; move to the rack
TRIGGER WHEN DISTANCE=1 DELAY=-1 DO Schrittmerker_R1Place(10150,10002,FPlace_R1_L2_S4_VP1,XPlace_R1_L2_S4_VP1) PRIO=-1
;FOLD PTP Place_R1_L2_S4_VP1 CONT Vel=12 % PPlace_R1_L2_S4_VP1 Tool[2]:Lower Gripper Base[0];%{PE}%R8.3.21,%MKUKATPBASIS,%CMOVE,%VPTP,%P 1:PTP, 2:Place_R1_L2_S4_VP1, 3:C_DIS, 5:12, 7:PPlace_R1_L2_S4_VP1
$BWDSTART=FALSE
PDAT_ACT= PPPlace_R1_L2_S4_VP1
FDAT_ACT= FPlace_R1_L2_S4_VP1
BAS(#PTP_PARAMS,12)
PTP XPlace_R1_L2_S4_VP1 C_DIS
;ENDFOLD
TRIGGER WHEN DISTANCE=1 DELAY=-1 DO Schrittmerker_R1Place(10151,10150,FPlace_R1_L2_S4_VP2,XPlace_R1_L2_S4_VP2) PRIO=-1
;FOLD PTP Place_R1_L2_S4_VP2 CONT Vel=12 % PPlace_R1_L2_S4_VP2 Tool[2]:Lower Gripper Base[0];%{PE}%R8.3.21,%MKUKATPBASIS,%CMOVE,%VPTP,%P 1:PTP, 2:Place_R1_L2_S4_VP2, 3:C_DIS, 5:12, 7:PPlace_R1_L2_S4_VP2
$BWDSTART=FALSE
PDAT_ACT= PPPlace_R1_L2_S4_VP2
FDAT_ACT= FPlace_R1_L2_S4_VP2
BAS(#PTP_PARAMS,12)
PTP XPlace_R1_L2_S4_VP2 C_DIS
;ENDFOLD
TRIGGER WHEN DISTANCE=1 DELAY=-1 DO Schrittmerker_R1Place(10152,10151,FPlace_R1_L2_S4_VP3,XPlace_R1_L2_S4_VP3) PRIO=-1
;FOLD PTP Place_R1_L2_S4_VP3 CONT Vel=12 % PPlace_R1_L2_S4_VP3 Tool[2]:Lower Gripper Base[0];%{PE}%R8.3.21,%MKUKATPBASIS,%CMOVE,%VPTP,%P 1:PTP, 2:Place_R1_L2_S4_VP3, 3:C_DIS, 5:12, 7:PPlace_R1_L2_S4_VP3
$BWDSTART=FALSE
PDAT_ACT= PPPlace_R1_L2_S4_VP3
FDAT_ACT= FPlace_R1_L2_S4_VP3
BAS(#PTP_PARAMS,12)
PTP XPlace_R1_L2_S4_VP3 C_DIS
;ENDFOLD
TRIGGER WHEN DISTANCE=1 DELAY=-1 DO Schrittmerker_R1Place(10153,10152,FPlace_R1_L2_S4_VP4,XPlace_R1_L2_S4_VP4) PRIO=-1
;FOLD PTP Place_R1_L2_S4_VP4 CONT Vel=12 % PPlace_R1_L2_S4_VP4 Tool[2]:Lower Gripper Base[0];%{PE}%R8.3.21,%MKUKATPBASIS,%CMOVE,%VPTP,%P 1:PTP, 2:Place_R1_L2_S4_VP4, 3:C_DIS, 5:12, 7:PPlace_R1_L2_S4_VP4
$BWDSTART=FALSE
PDAT_ACT= PPPlace_R1_L2_S4_VP4
FDAT_ACT= FPlace_R1_L2_S4_VP4
BAS(#PTP_PARAMS,12)
PTP XPlace_R1_L2_S4_VP4 C_DIS
;ENDFOLD
TRIGGER WHEN DISTANCE=1 DELAY=-1 DO Schrittmerker_R1Place(10154,10153,FPlace_R1_L2_S4_VP5,XPlace_R1_L2_S4_VP5) PRIO=-1
;FOLD PTP Place_R1_L2_S4_VP5 CONT Vel=12 % PPlace_R1_L2_S4_VP5 Tool[2]:Lower Gripper Base[1]:Rack1;%{PE}%R8.3.21,%MKUKATPBASIS,%CMOVE,%VPTP,%P 1:PTP, 2:Place_R1_L2_S4_VP5, 3:C_DIS, 5:12, 7:PPlace_R1_L2_S4_VP5
$BWDSTART=FALSE
PDAT_ACT= PPPlace_R1_L2_S4_VP5
FDAT_ACT= FPlace_R1_L2_S4_VP5
BAS(#PTP_PARAMS,12)
PTP XPlace_R1_L2_S4_VP5 C_DIS
;ENDFOLD

TRIGGER WHEN DISTANCE=1 DELAY=-1 DO Schrittmerker_R1Place(10155,10154,FPlace_R1_L2_S4_Check,XPlace_R1_L2_S4_Check) PRIO=-1
;FOLD PTP Place_R1_L2_S4_Check Vel=12 % PPlace_R1_L2_S4_Check Tool[2]:Lower Gripper Base[1]:Rack1;%{PE}%R8.3.21,%MKUKATPBASIS,%CMOVE,%VPTP,%P 1:PTP, 2:Place_R1_L2_S4_Check, 3:, 5:12, 7:PPlace_R1_L2_S4_Check
$BWDSTART=FALSE
PDAT_ACT= PPPlace_R1_L2_S4_Check
FDAT_ACT= FPlace_R1_L2_S4_Check
BAS(#PTP_PARAMS,12)
PTP XPlace_R1_L2_S4_Check
;ENDFOLD

;***************************************************
;FOLD Pruefe Platz frei
IF (DetectPart(CHECK_SHELF,PLACE)==OCCUPIED) THEN
  UP_Rueckzug_R1Place( )
  RETURN
ENDIF
;ENDFOLD
;***************************************************

TRIGGER WHEN DISTANCE=1 DELAY=-1 DO Schrittmerker_R1Place(10156,10155,FPlace_R1_L2_S4_VP6,XPlace_R1_L2_S4_VP6) PRIO=-1
;FOLD LIN Place_R1_L2_S4_VP6 CONT Vel=0.5 m/s LPlace_R1_L2_S4_VP6 Tool[2]:Lower Gripper Base[1]:Rack1;%{PE}%R8.3.21,%MKUKATPBASIS,%CMOVE,%VLIN,%P 1:LIN, 2:Place_R1_L2_S4_VP6, 3:C_DIS C_DIS, 5:0.5, 7:LPlace_R1_L2_S4_VP6
$BWDSTART=FALSE
LDAT_ACT= LLPlace_R1_L2_S4_VP6
FDAT_ACT= FPlace_R1_L2_S4_VP6
BAS(#CP_PARAMS,0.5)
LIN XPlace_R1_L2_S4_VP6 C_DIS C_DIS
;ENDFOLD
TRIGGER WHEN DISTANCE=1 DELAY=-1 DO Schrittmerker_R1Place(10157,10156,FPlace_R1_L2_S4_VP7,XPlace_R1_L2_S4_VP7) PRIO=-1
;FOLD LIN Place_R1_L2_S4_VP7 CONT Vel=0.5 m/s LPlace_R1_L2_S4_VP7 Tool[2]:Lower Gripper Base[1]:Rack1;%{PE}%R8.3.21,%MKUKATPBASIS,%CMOVE,%VLIN,%P 1:LIN, 2:Place_R1_L2_S4_VP7, 3:C_DIS C_DIS, 5:0.5, 7:LPlace_R1_L2_S4_VP7
$BWDSTART=FALSE
LDAT_ACT= LLPlace_R1_L2_S4_VP7
FDAT_ACT= FPlace_R1_L2_S4_VP7
BAS(#CP_PARAMS,0.5)
LIN XPlace_R1_L2_S4_VP7 C_DIS C_DIS
;ENDFOLD

;FOLD Test the way back home - part 1
CONTINUE
IF ($FLAG[M_Test_GrdstFahren1] AND NOT $FLAG[M_Test_GrdstFahren2]) THEN
  $FLAG[M_Test_GrdstFahren2]=TRUE
  UP_Rueckzug( )
  RETURN
ENDIF
;ENDFOLD

;-------------------------------
; Place part position
;-------------------------------
TRIGGER WHEN DISTANCE=1 DELAY=-1 DO Schrittmerker_R1Place(10158,10159,FPlace_R1_L2_S4_AP,XPlace_R1_L2_S4_AP) PRIO=-1
;FOLD LIN Place_R1_L2_S4_AP Vel=0.2 m/s LPlace_R1_L2_S4_AP Tool[2]:Lower Gripper Base[1]:Rack1;%{PE}%R8.3.21,%MKUKATPBASIS,%CMOVE,%VLIN,%P 1:LIN, 2:Place_R1_L2_S4_AP, 3:, 5:0.2, 7:LPlace_R1_L2_S4_AP
$BWDSTART=FALSE
LDAT_ACT= LLPlace_R1_L2_S4_AP
FDAT_ACT= FPlace_R1_L2_S4_AP
BAS(#CP_PARAMS,0.2)
LIN XPlace_R1_L2_S4_AP
;ENDFOLD

;FOLD Test the way back home - part 2
CONTINUE
IF $FLAG[M_Test_GrdstFahren2] THEN
  $FLAG[M_Test_GrdstFahren2]=FALSE
  UP_Rueckzug( )
  RETURN
ENDIF
;ENDFOLD

;***************************************************
; Disable part lost detection
SetPartLostDetection(NO_PART)
;***************************************************

TRIGGER WHEN DISTANCE=1 DELAY=-1 DO Schrittmerker_R1Place(10159,10160,FPlace_R1_L2_S4_NP1,XPlace_R1_L2_S4_NP1) PRIO=-1
;FOLD LIN Place_R1_L2_S4_NP1 Vel=0.2 m/s LPlace_R1_L2_S4_NP1 Tool[2]:Lower Gripper Base[1]:Rack1;%{PE}%R8.3.21,%MKUKATPBASIS,%CMOVE,%VLIN,%P 1:LIN, 2:Place_R1_L2_S4_NP1, 3:C_DIS C_DIS, 5:0.2, 7:LPlace_R1_L2_S4_NP1
$BWDSTART=FALSE
LDAT_ACT= LLPlace_R1_L2_S4_NP1
FDAT_ACT= FPlace_R1_L2_S4_NP1
BAS(#CP_PARAMS,0.2)
LIN XPlace_R1_L2_S4_NP1
;ENDFOLD

;***************************************************
; Check for part present (empty gripper)
CheckPartPresent(EMPTY_GRIPPER)
;***************************************************
; set load data
SetLoadData( )
;***************************************************

TRIGGER WHEN DISTANCE=1 DELAY=-1 DO Schrittmerker_R1Place(10160,10161,FPlace_R1_L2_S4_NP2,XPlace_R1_L2_S4_NP2) PRIO=-1
;FOLD LIN Place_R1_L2_S4_NP2 CONT Vel=0.5 m/s LPlace_R1_L2_S4_NP2 Tool[2]:Lower Gripper Base[1]:Rack1;%{PE}%R8.3.21,%MKUKATPBASIS,%CMOVE,%VLIN,%P 1:LIN, 2:Place_R1_L2_S4_NP2, 3:C_DIS C_DIS, 5:0.5, 7:LPlace_R1_L2_S4_NP2
$BWDSTART=FALSE
LDAT_ACT= LLPlace_R1_L2_S4_NP2
FDAT_ACT= FPlace_R1_L2_S4_NP2
BAS(#CP_PARAMS,0.5)
LIN XPlace_R1_L2_S4_NP2 C_DIS C_DIS
;ENDFOLD
TRIGGER WHEN DISTANCE=1 DELAY=-1 DO Schrittmerker_R1Place(10161,10162,FPlace_R1_L2_S4_NP3,XPlace_R1_L2_S4_NP3) PRIO=-1
;FOLD LIN Place_R1_L2_S4_NP3 Vel=0.5 m/s LPlace_R1_L2_S4_NP3 Tool[2]:Lower Gripper Base[1]:Rack 1 ;%{PE}
$BWDSTART=FALSE
LDAT_ACT= LLPlace_R1_L2_S4_NP3
FDAT_ACT= FPlace_R1_L2_S4_NP3
BAS(#CP_PARAMS,0.5)
LIN XPlace_R1_L2_S4_NP3
;ENDFOLD
TRIGGER WHEN DISTANCE=1 DELAY=-1 DO Schrittmerker_R1Place(10162,10163,FPlace_R1_L2_S4_NP4,XPlace_R1_L2_S4_NP4) PRIO=-1
;FOLD PTP Place_R1_L2_S4_NP4 CONT Vel=100 % PPlace_R1_L2_S4_NP4 Tool[2]:Lower Gripper Base[0];%{PE}%R8.3.21,%MKUKATPBASIS,%CMOVE,%VPTP,%P 1:PTP, 2:Place_R1_L2_S4_NP4, 3:C_DIS, 5:100, 7:PPlace_R1_L2_S4_NP4
$BWDSTART=FALSE
PDAT_ACT= PPPlace_R1_L2_S4_NP4
FDAT_ACT= FPlace_R1_L2_S4_NP4
BAS(#PTP_PARAMS,100)
PTP XPlace_R1_L2_S4_NP4 C_DIS
;ENDFOLD
TRIGGER WHEN DISTANCE=1 DELAY=-1 DO Schrittmerker_R1Place(10163,10164,FPlace_R1_L2_S4_NP5,XPlace_R1_L2_S4_NP5) PRIO=-1
;FOLD PTP Place_R1_L2_S4_NP5 CONT Vel=100 % PPlace_R1_L2_S4_NP5 Tool[2]:Lower Gripper Base[0];%{PE}%R8.3.21,%MKUKATPBASIS,%CMOVE,%VPTP,%P 1:PTP, 2:Place_R1_L2_S4_NP5, 3:C_DIS, 5:100, 7:PPlace_R1_L2_S4_NP5
$BWDSTART=FALSE
PDAT_ACT= PPPlace_R1_L2_S4_NP5
FDAT_ACT= FPlace_R1_L2_S4_NP5
BAS(#PTP_PARAMS,100)
PTP XPlace_R1_L2_S4_NP5 C_DIS
;ENDFOLD
TRIGGER WHEN DISTANCE=1 DELAY=-1 DO Schrittmerker_R1Place(10164,10165,FPlace_R1_L2_S4_NP6,XPlace_R1_L2_S4_NP6) PRIO=-1
;FOLD PTP Place_R1_L2_S4_NP6 CONT Vel=100 % PPlace_R1_L2_S4_NP6 Tool[2]:Lower Gripper Base[0];%{PE}%R8.3.21,%MKUKATPBASIS,%CMOVE,%VPTP,%P 1:PTP, 2:Place_R1_L2_S4_NP6, 3:C_DIS, 5:100, 7:PPlace_R1_L2_S4_NP6
$BWDSTART=FALSE
PDAT_ACT= PPPlace_R1_L2_S4_NP6
FDAT_ACT= FPlace_R1_L2_S4_NP6
BAS(#PTP_PARAMS,100)
PTP XPlace_R1_L2_S4_NP6 C_DIS
;ENDFOLD
TRIGGER WHEN DISTANCE=1 DELAY=-1 DO Schrittmerker_R1Place(10165,10166,FPlace_R1_L2_S4_NP7,XPlace_R1_L2_S4_NP7) PRIO=-1
;FOLD PTP Place_R1_L2_S4_NP7 CONT Vel=100 % PPlace_R1_L2_S4_NP7 Tool[2]:Lower Gripper Base[0];%{PE}%R8.3.21,%MKUKATPBASIS,%CMOVE,%VPTP,%P 1:PTP, 2:Place_R1_L2_S4_NP7, 3:C_DIS, 5:100, 7:PPlace_R1_L2_S4_NP7
$BWDSTART=FALSE
PDAT_ACT= PPPlace_R1_L2_S4_NP7
FDAT_ACT= FPlace_R1_L2_S4_NP7
BAS(#PTP_PARAMS,100)
PTP XPlace_R1_L2_S4_NP7 C_DIS
;ENDFOLD
TRIGGER WHEN DISTANCE=1 DELAY=-1 DO Schrittmerker_R1Place(10166,10167,FPlace_R1_L2_S4_NP8,XPlace_R1_L2_S4_NP8) PRIO=-1
;FOLD PTP Place_R1_L2_S4_NP8 CONT Vel=100 % PPlace_R1_L2_S4_NP8 Tool[2]:Lower Gripper Base[0];%{PE}%R8.3.21,%MKUKATPBASIS,%CMOVE,%VPTP,%P 1:PTP, 2:Place_R1_L2_S4_NP8, 3:C_DIS, 5:100, 7:PPlace_R1_L2_S4_NP8
$BWDSTART=FALSE
PDAT_ACT= PPPlace_R1_L2_S4_NP8
FDAT_ACT= FPlace_R1_L2_S4_NP8
BAS(#PTP_PARAMS,100)
PTP XPlace_R1_L2_S4_NP8 C_DIS
;ENDFOLD

TRIGGER WHEN DISTANCE=1 DELAY=-1 DO Schrittmerker_R1Place(10167,10002,FHOME1,$nullframe,XHOME1) PRIO=-1
;FOLD PTP HOME1 Vel=100 % PHome1;%{PE}%R8.3.21,%MKUKATPBASIS,%CMOVE,%VPTP,%P 1:PTP, 2:HOME1, 3:, 5:100, 7:PHome1
$BWDSTART=FALSE
PDAT_ACT= PPHome1
FDAT_ACT= FHOME1
BAS(#PTP_PARAMS,100)
PTP XHOME1
;ENDFOLD

;***************************************************
;FOLD Final tasks.
; Robot out of area Rack 1 Level 2
RobAusStorage1_2_A68=RESET_IN_AREA
;***************************************************
; stop cyclic clearence check
$CYCFLAG[ciFreigabeSPS]=DISABLE_MONITORING
;***************************************************
; Disable collision detection
;FOLD COLLDETECT Off ;%{PE}
;FOLD Parameters ;%{h}
;Params IlfProvider=kukaroboter.basistech.inlineforms.colldetect.off; CollDetect.Command=Off
;ENDFOLD
USE_CD_PARAMS(0)
;ENDFOLD
;***************************************************
;ENDFOLD
;***************************************************

END

; ##################################################

GLOBAL DEF UP_Place_R1_L3_S1( )
;***************************************************
; Place part on:
;    Rack  1
;    Level 3
;    Shelf 1
;***************************************************
;FOLD Preconditions - Vorraussetzungen
;***************************************************
; Enable collision detection
;FOLD COLLDETECT SetLimits Axis1: 150 % Axis2: 200 % Axis3: 150 % Axis4: 200 % Axis5: 150 % Axis6: 150 % ;%{PE}
;FOLD Parameters ;%{h}
;Params IlfProvider=kukaroboter.basistech.inlineforms.colldetect.setlimits; CollDetect.Command=SetLimits; CollDetect.Axis1=150; CollDetect.Axis2=200; CollDetect.Axis3=150; CollDetect.Axis4=200; CollDetect.Axis5=150; CollDetect.Axis6=150
;ENDFOLD
SET_TQ_VALUES(150, 200, 150, 200, 150, 150)
;ENDFOLD
;***************************************************
; Check for part in gripper (tool 2).
CheckPartPresent(OCCUPIED_GRIPPER,PART_ON_TOOL_2)
;***************************************************
; Enable part lost detection for tool 2
SetPartLostDetection(PART_ON_TOOL_2)
;***************************************************
; Set load data.
SetLoadData( )
;***************************************************
; Robot has to start from home position.
IF NOT $IN_HOME1 THEN
  UP_HomeToHome(1)
ENDIF
;***************************************************
;ENDFOLD

TRIGGER WHEN DISTANCE=1 DELAY=-1 DO Schrittmerker_R1Place(10002,10002,FHOME1,$nullframe,XHOME1) PRIO=-1
;FOLD PTP HOME1 Vel=12 % PHome1;%{PE}%R8.3.21,%MKUKATPBASIS,%CMOVE,%VPTP,%P 1:PTP, 2:HOME1, 3:, 5:12, 7:PHome1
$BWDSTART=FALSE
PDAT_ACT= PPHome1
FDAT_ACT= FHOME1
BAS(#PTP_PARAMS,12)
PTP XHOME1
;ENDFOLD

;***************************************************
;FOLD Area clearence handshake.
IF NOT $FLAG[M_Inbetriebnahme] THEN
  ;-------------------------------------------------
  ; Request area clearence.
  AnfStoer_Store1_3_A101=SET_REQUEST
  ;-------------------------------------------------
  ; Wait for area clearence from PLC.
  WAIT_FOR_INPUT("Frg_Storage1_3_E69",TRUE)
  ;-------------------------------------------------
  ; Reset area clearence request.
  AnfStoer_Store1_3_A101=RESET_REQUEST
  ;-------------------------------------------------
  ; start cyclic clearence check
  $CYCFLAG[ciFreigabeSPS]=Frg_Storage1_3_E69
  ;-------------------------------------------------
ENDIF
;***************************************************
; set "robot in area"
RobAusStorage1_3_A69=SET_IN_AREA
;ENDFOLD
;***************************************************

;***************************************************
;FOLD Check for Teachmode
IF $FLAG[M_Teachen] THEN
  WAIT FOR $T1
ENDIF
;ENDFOLD
;***************************************************

; move to the rack
TRIGGER WHEN DISTANCE=1 DELAY=-1 DO Schrittmerker_R1Place(10170,10002,FPlace_R1_L3_S1_VP1,XPlace_R1_L3_S1_VP1) PRIO=-1
;FOLD PTP Place_R1_L3_S1_VP1 CONT Vel=12 % PPlace_R1_L3_S1_VP1 Tool[2]:Lower Gripper Base[0];%{PE}%R8.3.21,%MKUKATPBASIS,%CMOVE,%VPTP,%P 1:PTP, 2:Place_R1_L3_S1_VP1, 3:C_DIS, 5:12, 7:PPlace_R1_L3_S1_VP1
$BWDSTART=FALSE
PDAT_ACT= PPPlace_R1_L3_S1_VP1
FDAT_ACT= FPlace_R1_L3_S1_VP1
BAS(#PTP_PARAMS,12)
PTP XPlace_R1_L3_S1_VP1 C_DIS
;ENDFOLD
TRIGGER WHEN DISTANCE=1 DELAY=-1 DO Schrittmerker_R1Place(10171,10170,FPlace_R1_L3_S1_VP2,XPlace_R1_L3_S1_VP2) PRIO=-1
;FOLD PTP Place_R1_L3_S1_VP2 CONT Vel=12 % PPlace_R1_L3_S1_VP2 Tool[2]:Lower Gripper Base[0];%{PE}%R8.3.21,%MKUKATPBASIS,%CMOVE,%VPTP,%P 1:PTP, 2:Place_R1_L3_S1_VP2, 3:C_DIS, 5:12, 7:PPlace_R1_L3_S1_VP2
$BWDSTART=FALSE
PDAT_ACT= PPPlace_R1_L3_S1_VP2
FDAT_ACT= FPlace_R1_L3_S1_VP2
BAS(#PTP_PARAMS,12)
PTP XPlace_R1_L3_S1_VP2 C_DIS
;ENDFOLD
TRIGGER WHEN DISTANCE=1 DELAY=-1 DO Schrittmerker_R1Place(10172,10171,FPlace_R1_L3_S1_VP3,XPlace_R1_L3_S1_VP3) PRIO=-1
;FOLD PTP Place_R1_L3_S1_VP3 CONT Vel=12 % PPlace_R1_L3_S1_VP3 Tool[2]:Lower Gripper Base[0];%{PE}%R8.3.21,%MKUKATPBASIS,%CMOVE,%VPTP,%P 1:PTP, 2:Place_R1_L3_S1_VP3, 3:C_DIS, 5:12, 7:PPlace_R1_L3_S1_VP3
$BWDSTART=FALSE
PDAT_ACT= PPPlace_R1_L3_S1_VP3
FDAT_ACT= FPlace_R1_L3_S1_VP3
BAS(#PTP_PARAMS,12)
PTP XPlace_R1_L3_S1_VP3 C_DIS
;ENDFOLD
TRIGGER WHEN DISTANCE=1 DELAY=-1 DO Schrittmerker_R1Place(10173,10172,FPlace_R1_L3_S1_VP4,XPlace_R1_L3_S1_VP4) PRIO=-1
;FOLD PTP Place_R1_L3_S1_VP4 CONT Vel=12 % PPlace_R1_L3_S1_VP4 Tool[2]:Lower Gripper Base[1]:Rack1;%{PE}%R8.3.21,%MKUKATPBASIS,%CMOVE,%VPTP,%P 1:PTP, 2:Place_R1_L3_S1_VP4, 3:C_DIS, 5:12, 7:PPlace_R1_L3_S1_VP4
$BWDSTART=FALSE
PDAT_ACT= PPPlace_R1_L3_S1_VP4
FDAT_ACT= FPlace_R1_L3_S1_VP4
BAS(#PTP_PARAMS,12)
PTP XPlace_R1_L3_S1_VP4 C_DIS
;ENDFOLD

TRIGGER WHEN DISTANCE=1 DELAY=-1 DO Schrittmerker_R1Place(10174,10173,FPlace_R1_L3_S1_Check,XPlace_R1_L3_S1_Check) PRIO=-1
;FOLD PTP Place_R1_L3_S1_Check Vel=12 % PPlace_R1_L3_S1_Check Tool[2]:Lower Gripper Base[1]:Rack1;%{PE}%R8.3.21,%MKUKATPBASIS,%CMOVE,%VPTP,%P 1:PTP, 2:Place_R1_L3_S1_Check, 3:, 5:12, 7:PPlace_R1_L3_S1_Check
$BWDSTART=FALSE
PDAT_ACT= PPPlace_R1_L3_S1_Check
FDAT_ACT= FPlace_R1_L3_S1_Check
BAS(#PTP_PARAMS,12)
PTP XPlace_R1_L3_S1_Check
;ENDFOLD

;***************************************************
;FOLD Pruefe Platz frei
IF (DetectPart(CHECK_SHELF,PLACE)==OCCUPIED) THEN
  UP_Rueckzug_R1Place( )
  RETURN
ENDIF
;ENDFOLD
;***************************************************

TRIGGER WHEN DISTANCE=1 DELAY=-1 DO Schrittmerker_R1Place(10175,10174,FPlace_R1_L3_S1_VP5,XPlace_R1_L3_S1_VP5) PRIO=-1
;FOLD LIN Place_R1_L3_S1_VP5 CONT Vel=0.5 m/s LPlace_R1_L3_S1_VP5 Tool[2]:Lower Gripper Base[1]:Rack1;%{PE}%R8.3.21,%MKUKATPBASIS,%CMOVE,%VLIN,%P 1:LIN, 2:Place_R1_L3_S1_VP5, 3:C_DIS C_DIS, 5:0.5, 7:LPlace_R1_L3_S1_VP5
$BWDSTART=FALSE
LDAT_ACT= LLPlace_R1_L3_S1_VP5
FDAT_ACT= FPlace_R1_L3_S1_VP5
BAS(#CP_PARAMS,0.5)
LIN XPlace_R1_L3_S1_VP5 C_DIS C_DIS
;ENDFOLD
TRIGGER WHEN DISTANCE=1 DELAY=-1 DO Schrittmerker_R1Place(10176,10175,FPlace_R1_L3_S1_VP6,XPlace_R1_L3_S1_VP6) PRIO=-1
;FOLD LIN Place_R1_L3_S1_VP6 CONT Vel=0.5 m/s LPlace_R1_L3_S1_VP6 Tool[2]:Lower Gripper Base[1]:Rack1;%{PE}%R8.3.21,%MKUKATPBASIS,%CMOVE,%VLIN,%P 1:LIN, 2:Place_R1_L3_S1_VP6, 3:C_DIS C_DIS, 5:0.5, 7:LPlace_R1_L3_S1_VP6
$BWDSTART=FALSE
LDAT_ACT= LLPlace_R1_L3_S1_VP6
FDAT_ACT= FPlace_R1_L3_S1_VP6
BAS(#CP_PARAMS,0.5)
LIN XPlace_R1_L3_S1_VP6 C_DIS C_DIS
;ENDFOLD
TRIGGER WHEN DISTANCE=1 DELAY=-1 DO Schrittmerker_R1Place(10177,10176,FPlace_R1_L3_S1_VP7,XPlace_R1_L3_S1_VP7) PRIO=-1
;FOLD LIN Place_R1_L3_S1_VP7 CONT Vel=0.5 m/s LPlace_R1_L3_S1_VP7 Tool[2]:Lower Gripper Base[1]:Rack1;%{PE}%R8.3.21,%MKUKATPBASIS,%CMOVE,%VLIN,%P 1:LIN, 2:Place_R1_L3_S1_VP7, 3:C_DIS C_DIS, 5:0.5, 7:LPlace_R1_L3_S1_VP7
$BWDSTART=FALSE
LDAT_ACT= LLPlace_R1_L3_S1_VP7
FDAT_ACT= FPlace_R1_L3_S1_VP7
BAS(#CP_PARAMS,0.5)
LIN XPlace_R1_L3_S1_VP7 C_DIS C_DIS
;ENDFOLD

;FOLD Test the way back home - part 1
CONTINUE
IF ($FLAG[M_Test_GrdstFahren1] AND NOT $FLAG[M_Test_GrdstFahren2]) THEN
  $FLAG[M_Test_GrdstFahren2]=TRUE
  UP_Rueckzug( )
  RETURN
ENDIF
;ENDFOLD

;-------------------------------
; Place part position
;-------------------------------
TRIGGER WHEN DISTANCE=1 DELAY=-1 DO Schrittmerker_R1Place(10178,10179,FPlace_R1_L3_S1_AP,XPlace_R1_L3_S1_AP) PRIO=-1
;FOLD LIN Place_R1_L3_S1_AP Vel=0.2 m/s LPlace_R1_L3_S1_AP Tool[2]:Lower Gripper Base[1]:Rack1;%{PE}%R8.3.21,%MKUKATPBASIS,%CMOVE,%VLIN,%P 1:LIN, 2:Place_R1_L3_S1_AP, 3:, 5:0.2, 7:LPlace_R1_L3_S1_AP
$BWDSTART=FALSE
LDAT_ACT= LLPlace_R1_L3_S1_AP
FDAT_ACT= FPlace_R1_L3_S1_AP
BAS(#CP_PARAMS,0.2)
LIN XPlace_R1_L3_S1_AP
;ENDFOLD

;FOLD Test the way back home - part 2
CONTINUE
IF $FLAG[M_Test_GrdstFahren2] THEN
  $FLAG[M_Test_GrdstFahren2]=FALSE
  UP_Rueckzug( )
  RETURN
ENDIF
;ENDFOLD

;***************************************************
; Disable part lost detection
SetPartLostDetection(NO_PART)
;***************************************************

TRIGGER WHEN DISTANCE=1 DELAY=-1 DO Schrittmerker_R1Place(10179,10180,FPlace_R1_L3_S1_NP1,XPlace_R1_L3_S1_NP1) PRIO=-1
;FOLD LIN Place_R1_L3_S1_NP1 Vel=0.2 m/s LPlace_R1_L3_S1_NP1 Tool[2]:Lower Gripper Base[1]:Rack1;%{PE}%R8.3.21,%MKUKATPBASIS,%CMOVE,%VLIN,%P 1:LIN, 2:Place_R1_L3_S1_NP1, 3:C_DIS C_DIS, 5:0.2, 7:LPlace_R1_L3_S1_NP1
$BWDSTART=FALSE
LDAT_ACT= LLPlace_R1_L3_S1_NP1
FDAT_ACT= FPlace_R1_L3_S1_NP1
BAS(#CP_PARAMS,0.2)
LIN XPlace_R1_L3_S1_NP1
;ENDFOLD

;***************************************************
; Check for part present (empty gripper)
CheckPartPresent(EMPTY_GRIPPER)
;***************************************************
; set load data
SetLoadData( )
;***************************************************

TRIGGER WHEN DISTANCE=1 DELAY=-1 DO Schrittmerker_R1Place(10180,10181,FPlace_R1_L3_S1_NP2,XPlace_R1_L3_S1_NP2) PRIO=-1
;FOLD LIN Place_R1_L3_S1_NP2 CONT Vel=0.5 m/s LPlace_R1_L3_S1_NP2 Tool[2]:Lower Gripper Base[1]:Rack1;%{PE}%R8.3.21,%MKUKATPBASIS,%CMOVE,%VLIN,%P 1:LIN, 2:Place_R1_L3_S1_NP2, 3:C_DIS C_DIS, 5:0.5, 7:LPlace_R1_L3_S1_NP2
$BWDSTART=FALSE
LDAT_ACT= LLPlace_R1_L3_S1_NP2
FDAT_ACT= FPlace_R1_L3_S1_NP2
BAS(#CP_PARAMS,0.5)
LIN XPlace_R1_L3_S1_NP2 C_DIS C_DIS
;ENDFOLD
TRIGGER WHEN DISTANCE=1 DELAY=-1 DO Schrittmerker_R1Place(10181,10182,FPlace_R1_L3_S1_NP3,XPlace_R1_L3_S1_NP3) PRIO=-1
;FOLD LIN Place_R1_L3_S1_NP3 CONT Vel=0.5 m/s LPlace_R1_L3_S1_NP3 Tool[2]:Lower Gripper Base[1]:Rack1;%{PE}%R8.3.21,%MKUKATPBASIS,%CMOVE,%VLIN,%P 1:LIN, 2:Place_R1_L3_S1_NP3, 3:C_DIS C_DIS, 5:0.5, 7:LPlace_R1_L3_S1_NP3
$BWDSTART=FALSE
LDAT_ACT= LLPlace_R1_L3_S1_NP3
FDAT_ACT= FPlace_R1_L3_S1_NP3
BAS(#CP_PARAMS,0.5)
LIN XPlace_R1_L3_S1_NP3 C_DIS C_DIS
;ENDFOLD
TRIGGER WHEN DISTANCE=1 DELAY=-1 DO Schrittmerker_R1Place(10182,10183,FPlace_R1_L3_S1_NP4,XPlace_R1_L3_S1_NP4) PRIO=-1
;FOLD LIN Place_R1_L3_S1_NP4 CONT Vel=0.5 m/s LPlace_R1_L3_S1_NP4 Tool[2]:Lower Gripper Base[1]:Rack1;%{PE}%R8.3.21,%MKUKATPBASIS,%CMOVE,%VLIN,%P 1:LIN, 2:Place_R1_L3_S1_NP4, 3:C_DIS C_DIS, 5:0.5, 7:LPlace_R1_L3_S1_NP4
$BWDSTART=FALSE
LDAT_ACT= LLPlace_R1_L3_S1_NP4
FDAT_ACT= FPlace_R1_L3_S1_NP4
BAS(#CP_PARAMS,0.5)
LIN XPlace_R1_L3_S1_NP4 C_DIS C_DIS
;ENDFOLD
TRIGGER WHEN DISTANCE=1 DELAY=-1 DO Schrittmerker_R1Place(10183,10184,FPlace_R1_L3_S1_NP5,XPlace_R1_L3_S1_NP5) PRIO=-1
;FOLD PTP Place_R1_L3_S1_NP5 CONT Vel=100 % PPlace_R1_L3_S1_NP5 Tool[2]:Lower Gripper Base[0];%{PE}%R8.3.21,%MKUKATPBASIS,%CMOVE,%VPTP,%P 1:PTP, 2:Place_R1_L3_S1_NP5, 3:C_DIS, 5:100, 7:PPlace_R1_L3_S1_NP5
$BWDSTART=FALSE
PDAT_ACT= PPPlace_R1_L3_S1_NP5
FDAT_ACT= FPlace_R1_L3_S1_NP5
BAS(#PTP_PARAMS,100)
PTP XPlace_R1_L3_S1_NP5 C_DIS
;ENDFOLD
TRIGGER WHEN DISTANCE=1 DELAY=-1 DO Schrittmerker_R1Place(10184,10185,FPlace_R1_L3_S1_NP6,XPlace_R1_L3_S1_NP6) PRIO=-1
;FOLD PTP Place_R1_L3_S1_NP6 CONT Vel=100 % PPlace_R1_L3_S1_NP6 Tool[2]:Lower Gripper Base[0];%{PE}%R8.3.21,%MKUKATPBASIS,%CMOVE,%VPTP,%P 1:PTP, 2:Place_R1_L3_S1_NP6, 3:C_DIS, 5:100, 7:PPlace_R1_L3_S1_NP6
$BWDSTART=FALSE
PDAT_ACT= PPPlace_R1_L3_S1_NP6
FDAT_ACT= FPlace_R1_L3_S1_NP6
BAS(#PTP_PARAMS,100)
PTP XPlace_R1_L3_S1_NP6 C_DIS
;ENDFOLD
TRIGGER WHEN DISTANCE=1 DELAY=-1 DO Schrittmerker_R1Place(10185,10186,FPlace_R1_L3_S1_NP7,XPlace_R1_L3_S1_NP7) PRIO=-1
;FOLD PTP Place_R1_L3_S1_NP7 CONT Vel=100 % PPlace_R1_L3_S1_NP7 Tool[2]:Lower Gripper Base[0];%{PE}%R8.3.21,%MKUKATPBASIS,%CMOVE,%VPTP,%P 1:PTP, 2:Place_R1_L3_S1_NP7, 3:C_DIS, 5:100, 7:PPlace_R1_L3_S1_NP7
$BWDSTART=FALSE
PDAT_ACT= PPPlace_R1_L3_S1_NP7
FDAT_ACT= FPlace_R1_L3_S1_NP7
BAS(#PTP_PARAMS,100)
PTP XPlace_R1_L3_S1_NP7 C_DIS
;ENDFOLD
TRIGGER WHEN DISTANCE=1 DELAY=-1 DO Schrittmerker_R1Place(10186,10187,FPlace_R1_L3_S1_NP8,XPlace_R1_L3_S1_NP8) PRIO=-1
;FOLD PTP Place_R1_L3_S1_NP8 CONT Vel=100 % PPlace_R1_L3_S1_NP8 Tool[2]:Lower Gripper Base[0];%{PE}%R8.3.21,%MKUKATPBASIS,%CMOVE,%VPTP,%P 1:PTP, 2:Place_R1_L3_S1_NP8, 3:C_DIS, 5:100, 7:PPlace_R1_L3_S1_NP8
$BWDSTART=FALSE
PDAT_ACT= PPPlace_R1_L3_S1_NP8
FDAT_ACT= FPlace_R1_L3_S1_NP8
BAS(#PTP_PARAMS,100)
PTP XPlace_R1_L3_S1_NP8 C_DIS
;ENDFOLD
TRIGGER WHEN DISTANCE=1 DELAY=-1 DO Schrittmerker_R1Place(10187,10188,FPlace_R1_L3_S1_NP9,XPlace_R1_L3_S1_NP9) PRIO=-1
;FOLD PTP Place_R1_L3_S1_NP9 CONT Vel=100 % PPlace_R1_L3_S1_NP9 Tool[2]:Lower Gripper Base[0];%{PE}%R8.3.21,%MKUKATPBASIS,%CMOVE,%VPTP,%P 1:PTP, 2:Place_R1_L3_S1_NP9, 3:C_DIS, 5:100, 7:PPlace_R1_L3_S1_NP9
$BWDSTART=FALSE
PDAT_ACT= PPPlace_R1_L3_S1_NP9
FDAT_ACT= FPlace_R1_L3_S1_NP9
BAS(#PTP_PARAMS,100)
PTP XPlace_R1_L3_S1_NP9 C_DIS
;ENDFOLD

TRIGGER WHEN DISTANCE=1 DELAY=-1 DO Schrittmerker_R1Place(10188,10002,FHOME1,$nullframe,XHOME1) PRIO=-1
;FOLD PTP HOME1 Vel=100 % PHome1;%{PE}%R8.3.21,%MKUKATPBASIS,%CMOVE,%VPTP,%P 1:PTP, 2:HOME1, 3:, 5:100, 7:PHome1
$BWDSTART=FALSE
PDAT_ACT= PPHome1
FDAT_ACT= FHOME1
BAS(#PTP_PARAMS,100)
PTP XHOME1
;ENDFOLD

;***************************************************
;FOLD Final tasks.
; Robot out of area Rack 1 Level 3
RobAusStorage1_3_A69=RESET_IN_AREA
;***************************************************
; stop cyclic clearence check
$CYCFLAG[ciFreigabeSPS]=DISABLE_MONITORING
;***************************************************
; Disable collision detection
;FOLD COLLDETECT Off ;%{PE}
;FOLD Parameters ;%{h}
;Params IlfProvider=kukaroboter.basistech.inlineforms.colldetect.off; CollDetect.Command=Off
;ENDFOLD
USE_CD_PARAMS(0)
;ENDFOLD
;***************************************************
;ENDFOLD
;***************************************************

END

; ##################################################

GLOBAL DEF UP_Place_R1_L3_S2( )
;***************************************************
; Place part on:
;    Rack  1
;    Level 3
;    Shelf 2
;***************************************************
;FOLD Preconditions - Vorraussetzungen
;***************************************************
; Enable collision detection
;FOLD COLLDETECT SetLimits Axis1: 150 % Axis2: 200 % Axis3: 150 % Axis4: 200 % Axis5: 150 % Axis6: 150 % ;%{PE}
;FOLD Parameters ;%{h}
;Params IlfProvider=kukaroboter.basistech.inlineforms.colldetect.setlimits; CollDetect.Command=SetLimits; CollDetect.Axis1=150; CollDetect.Axis2=200; CollDetect.Axis3=150; CollDetect.Axis4=200; CollDetect.Axis5=150; CollDetect.Axis6=150
;ENDFOLD
SET_TQ_VALUES(150, 200, 150, 200, 150, 150)
;ENDFOLD
;***************************************************
; Check for part in gripper (tool 2).
CheckPartPresent(OCCUPIED_GRIPPER,PART_ON_TOOL_2)
;***************************************************
; Enable part lost detection for tool 2
SetPartLostDetection(PART_ON_TOOL_2)
;***************************************************
; Set load data.
SetLoadData( )
;***************************************************
; Robot has to start from home position.
IF NOT $IN_HOME1 THEN
  UP_HomeToHome(1)
ENDIF
;***************************************************
;ENDFOLD

TRIGGER WHEN DISTANCE=1 DELAY=-1 DO Schrittmerker_R1Place(10002,10002,FHOME1,$nullframe,XHOME1) PRIO=-1
;FOLD PTP HOME1 Vel=12 % PHome1;%{PE}%R8.3.21,%MKUKATPBASIS,%CMOVE,%VPTP,%P 1:PTP, 2:HOME1, 3:, 5:12, 7:PHome1
$BWDSTART=FALSE
PDAT_ACT= PPHome1
FDAT_ACT= FHOME1
BAS(#PTP_PARAMS,12)
PTP XHOME1
;ENDFOLD

;***************************************************
;FOLD Area clearence handshake.
IF NOT $FLAG[M_Inbetriebnahme] THEN
  ;-------------------------------------------------
  ; Request area clearence.
  AnfStoer_Store1_3_A101=SET_REQUEST
  ;-------------------------------------------------
  ; Wait for area clearence from PLC.
  WAIT_FOR_INPUT("Frg_Storage1_3_E69",TRUE)
  ;-------------------------------------------------
  ; Reset area clearence request.
  AnfStoer_Store1_3_A101=RESET_REQUEST
  ;-------------------------------------------------
  ; start cyclic clearence check
  $CYCFLAG[ciFreigabeSPS]=Frg_Storage1_3_E69
  ;-------------------------------------------------
ENDIF
;***************************************************
; set "robot in area"
RobAusStorage1_3_A69=SET_IN_AREA
;ENDFOLD
;***************************************************

;***************************************************
;FOLD Check for Teachmode
IF $FLAG[M_Teachen] THEN
  WAIT FOR $T1
ENDIF
;ENDFOLD
;***************************************************

; move to the rack
TRIGGER WHEN DISTANCE=1 DELAY=-1 DO Schrittmerker_R1Place(10190,10002,FPlace_R1_L3_S2_VP1,XPlace_R1_L3_S2_VP1) PRIO=-1
;FOLD PTP Place_R1_L3_S2_VP1 CONT Vel=12 % PPlace_R1_L3_S2_VP1 Tool[2]:Lower Gripper Base[0];%{PE}%R8.3.21,%MKUKATPBASIS,%CMOVE,%VPTP,%P 1:PTP, 2:Place_R1_L3_S2_VP1, 3:C_DIS, 5:12, 7:PPlace_R1_L3_S2_VP1
$BWDSTART=FALSE
PDAT_ACT= PPPlace_R1_L3_S2_VP1
FDAT_ACT= FPlace_R1_L3_S2_VP1
BAS(#PTP_PARAMS,12)
PTP XPlace_R1_L3_S2_VP1 C_DIS
;ENDFOLD
TRIGGER WHEN DISTANCE=1 DELAY=-1 DO Schrittmerker_R1Place(10191,10190,FPlace_R1_L3_S2_VP2,XPlace_R1_L3_S2_VP2) PRIO=-1
;FOLD PTP Place_R1_L3_S2_VP2 CONT Vel=12 % PPlace_R1_L3_S2_VP2 Tool[2]:Lower Gripper Base[0];%{PE}%R8.3.21,%MKUKATPBASIS,%CMOVE,%VPTP,%P 1:PTP, 2:Place_R1_L3_S2_VP2, 3:C_DIS, 5:12, 7:PPlace_R1_L3_S2_VP2
$BWDSTART=FALSE
PDAT_ACT= PPPlace_R1_L3_S2_VP2
FDAT_ACT= FPlace_R1_L3_S2_VP2
BAS(#PTP_PARAMS,12)
PTP XPlace_R1_L3_S2_VP2 C_DIS
;ENDFOLD
TRIGGER WHEN DISTANCE=1 DELAY=-1 DO Schrittmerker_R1Place(10192,10191,FPlace_R1_L3_S2_VP3,XPlace_R1_L3_S2_VP3) PRIO=-1
;FOLD PTP Place_R1_L3_S2_VP3 CONT Vel=12 % PPlace_R1_L3_S2_VP3 Tool[2]:Lower Gripper Base[0];%{PE}%R8.3.21,%MKUKATPBASIS,%CMOVE,%VPTP,%P 1:PTP, 2:Place_R1_L3_S2_VP3, 3:C_DIS, 5:12, 7:PPlace_R1_L3_S2_VP3
$BWDSTART=FALSE
PDAT_ACT= PPPlace_R1_L3_S2_VP3
FDAT_ACT= FPlace_R1_L3_S2_VP3
BAS(#PTP_PARAMS,12)
PTP XPlace_R1_L3_S2_VP3 C_DIS
;ENDFOLD
TRIGGER WHEN DISTANCE=1 DELAY=-1 DO Schrittmerker_R1Place(10193,10192,FPlace_R1_L3_S2_VP4,XPlace_R1_L3_S2_VP4) PRIO=-1
;FOLD PTP Place_R1_L3_S2_VP4 CONT Vel=12 % PPlace_R1_L3_S2_VP4 Tool[2]:Lower Gripper Base[0];%{PE}%R8.3.21,%MKUKATPBASIS,%CMOVE,%VPTP,%P 1:PTP, 2:Place_R1_L3_S2_VP4, 3:C_DIS, 5:12, 7:PPlace_R1_L3_S2_VP4
$BWDSTART=FALSE
PDAT_ACT= PPPlace_R1_L3_S2_VP4
FDAT_ACT= FPlace_R1_L3_S2_VP4
BAS(#PTP_PARAMS,12)
PTP XPlace_R1_L3_S2_VP4 C_DIS
;ENDFOLD
TRIGGER WHEN DISTANCE=1 DELAY=-1 DO Schrittmerker_R1Place(10194,10193,FPlace_R1_L3_S2_VP5,XPlace_R1_L3_S2_VP5) PRIO=-1
;FOLD PTP Place_R1_L3_S2_VP5 CONT Vel=12 % PPlace_R1_L3_S2_VP5 Tool[2]:Lower Gripper Base[1]:Rack1;%{PE}%R8.3.21,%MKUKATPBASIS,%CMOVE,%VPTP,%P 1:PTP, 2:Place_R1_L3_S2_VP5, 3:C_DIS, 5:12, 7:PPlace_R1_L3_S2_VP5
$BWDSTART=FALSE
PDAT_ACT= PPPlace_R1_L3_S2_VP5
FDAT_ACT= FPlace_R1_L3_S2_VP5
BAS(#PTP_PARAMS,12)
PTP XPlace_R1_L3_S2_VP5 C_DIS
;ENDFOLD

TRIGGER WHEN DISTANCE=1 DELAY=-1 DO Schrittmerker_R1Place(10195,10194,FPlace_R1_L3_S2_Check,XPlace_R1_L3_S2_Check) PRIO=-1
;FOLD PTP Place_R1_L3_S2_Check Vel=12 % PPlace_R1_L3_S2_Check Tool[2]:Lower Gripper Base[1]:Rack1;%{PE}%R8.3.21,%MKUKATPBASIS,%CMOVE,%VPTP,%P 1:PTP, 2:Place_R1_L3_S2_Check, 3:, 5:12, 7:PPlace_R1_L3_S2_Check
$BWDSTART=FALSE
PDAT_ACT= PPPlace_R1_L3_S2_Check
FDAT_ACT= FPlace_R1_L3_S2_Check
BAS(#PTP_PARAMS,12)
PTP XPlace_R1_L3_S2_Check
;ENDFOLD

;***************************************************
;FOLD Pruefe Platz frei
IF (DetectPart(CHECK_SHELF,PLACE)==OCCUPIED) THEN
  UP_Rueckzug_R1Place( )
  RETURN
ENDIF
;ENDFOLD
;***************************************************

TRIGGER WHEN DISTANCE=1 DELAY=-1 DO Schrittmerker_R1Place(10196,10195,FPlace_R1_L3_S2_VP6,XPlace_R1_L3_S2_VP6) PRIO=-1
;FOLD LIN Place_R1_L3_S2_VP6 CONT Vel=0.5 m/s LPlace_R1_L3_S2_VP6 Tool[2]:Lower Gripper Base[1]:Rack1;%{PE}%R8.3.21,%MKUKATPBASIS,%CMOVE,%VLIN,%P 1:LIN, 2:Place_R1_L3_S2_VP6, 3:C_DIS C_DIS, 5:0.5, 7:LPlace_R1_L3_S2_VP6
$BWDSTART=FALSE
LDAT_ACT= LLPlace_R1_L3_S2_VP6
FDAT_ACT= FPlace_R1_L3_S2_VP6
BAS(#CP_PARAMS,0.5)
LIN XPlace_R1_L3_S2_VP6 C_DIS C_DIS
;ENDFOLD

;FOLD Test the way back home - part 1
CONTINUE
IF ($FLAG[M_Test_GrdstFahren1] AND NOT $FLAG[M_Test_GrdstFahren2]) THEN
  $FLAG[M_Test_GrdstFahren2]=TRUE
  UP_Rueckzug( )
  RETURN
ENDIF
;ENDFOLD

;-------------------------------
; Place part position
;-------------------------------
TRIGGER WHEN DISTANCE=1 DELAY=-1 DO Schrittmerker_R1Place(10197,10198,FPlace_R1_L3_S2_AP,XPlace_R1_L3_S2_AP) PRIO=-1
;FOLD LIN Place_R1_L3_S2_AP Vel=0.2 m/s LPlace_R1_L3_S2_AP Tool[2]:Lower Gripper Base[1]:Rack1;%{PE}%R8.3.21,%MKUKATPBASIS,%CMOVE,%VLIN,%P 1:LIN, 2:Place_R1_L3_S2_AP, 3:, 5:0.2, 7:LPlace_R1_L3_S2_AP
$BWDSTART=FALSE
LDAT_ACT= LLPlace_R1_L3_S2_AP
FDAT_ACT= FPlace_R1_L3_S2_AP
BAS(#CP_PARAMS,0.2)
LIN XPlace_R1_L3_S2_AP
;ENDFOLD

;FOLD Test the way back home - part 2
CONTINUE
IF $FLAG[M_Test_GrdstFahren2] THEN
  $FLAG[M_Test_GrdstFahren2]=FALSE
  UP_Rueckzug( )
  RETURN
ENDIF
;ENDFOLD

;***************************************************
; Disable part lost detection
SetPartLostDetection(NO_PART)
;***************************************************

TRIGGER WHEN DISTANCE=1 DELAY=-1 DO Schrittmerker_R1Place(10198,10199,FPlace_R1_L3_S2_NP1,XPlace_R1_L3_S2_NP1) PRIO=-1
;FOLD LIN Place_R1_L3_S2_NP1 Vel=0.2 m/s LPlace_R1_L3_S2_NP1 Tool[2]:Lower Gripper Base[1]:Rack1;%{PE}%R8.3.21,%MKUKATPBASIS,%CMOVE,%VLIN,%P 1:LIN, 2:Place_R1_L3_S2_NP1, 3:C_DIS C_DIS, 5:0.2, 7:LPlace_R1_L3_S2_NP1
$BWDSTART=FALSE
LDAT_ACT= LLPlace_R1_L3_S2_NP1
FDAT_ACT= FPlace_R1_L3_S2_NP1
BAS(#CP_PARAMS,0.2)
LIN XPlace_R1_L3_S2_NP1
;ENDFOLD

;***************************************************
; Check for part present (empty gripper)
CheckPartPresent(EMPTY_GRIPPER)
;***************************************************
; set load data
SetLoadData( )
;***************************************************

TRIGGER WHEN DISTANCE=1 DELAY=-1 DO Schrittmerker_R1Place(10199,10200,FPlace_R1_L3_S2_NP2,XPlace_R1_L3_S2_NP2) PRIO=-1
;FOLD LIN Place_R1_L3_S2_NP2 CONT Vel=0.5 m/s LPlace_R1_L3_S2_NP2 Tool[2]:Lower Gripper Base[1]:Rack1;%{PE}%R8.3.21,%MKUKATPBASIS,%CMOVE,%VLIN,%P 1:LIN, 2:Place_R1_L3_S2_NP2, 3:C_DIS C_DIS, 5:0.5, 7:LPlace_R1_L3_S2_NP2
$BWDSTART=FALSE
LDAT_ACT= LLPlace_R1_L3_S2_NP2
FDAT_ACT= FPlace_R1_L3_S2_NP2
BAS(#CP_PARAMS,0.5)
LIN XPlace_R1_L3_S2_NP2 C_DIS C_DIS
;ENDFOLD
TRIGGER WHEN DISTANCE=1 DELAY=-1 DO Schrittmerker_R1Place(10200,10201,FPlace_R1_L3_S2_NP3,XPlace_R1_L3_S2_NP3) PRIO=-1
;FOLD PTP Place_R1_L3_S2_NP3 CONT Vel=100 % PPlace_R1_L3_S2_NP3 Tool[2]:Lower Gripper Base[0];%{PE}%R8.3.21,%MKUKATPBASIS,%CMOVE,%VPTP,%P 1:PTP, 2:Place_R1_L3_S2_NP3, 3:C_DIS, 5:100, 7:PPlace_R1_L3_S2_NP3
$BWDSTART=FALSE
PDAT_ACT= PPPlace_R1_L3_S2_NP3
FDAT_ACT= FPlace_R1_L3_S2_NP3
BAS(#PTP_PARAMS,100)
PTP XPlace_R1_L3_S2_NP3 C_DIS
;ENDFOLD
TRIGGER WHEN DISTANCE=1 DELAY=-1 DO Schrittmerker_R1Place(10201,10202,FPlace_R1_L3_S2_NP4,XPlace_R1_L3_S2_NP4) PRIO=-1
;FOLD PTP Place_R1_L3_S2_NP4 CONT Vel=100 % PPlace_R1_L3_S2_NP4 Tool[2]:Lower Gripper Base[0];%{PE}%R8.3.21,%MKUKATPBASIS,%CMOVE,%VPTP,%P 1:PTP, 2:Place_R1_L3_S2_NP4, 3:C_DIS, 5:100, 7:PPlace_R1_L3_S2_NP4
$BWDSTART=FALSE
PDAT_ACT= PPPlace_R1_L3_S2_NP4
FDAT_ACT= FPlace_R1_L3_S2_NP4
BAS(#PTP_PARAMS,100)
PTP XPlace_R1_L3_S2_NP4 C_DIS
;ENDFOLD
TRIGGER WHEN DISTANCE=1 DELAY=-1 DO Schrittmerker_R1Place(10202,10203,FPlace_R1_L3_S2_NP5,XPlace_R1_L3_S2_NP5) PRIO=-1
;FOLD PTP Place_R1_L3_S2_NP5 CONT Vel=100 % PPlace_R1_L3_S2_NP5 Tool[2]:Lower Gripper Base[0];%{PE}%R8.3.21,%MKUKATPBASIS,%CMOVE,%VPTP,%P 1:PTP, 2:Place_R1_L3_S2_NP5, 3:C_DIS, 5:100, 7:PPlace_R1_L3_S2_NP5
$BWDSTART=FALSE
PDAT_ACT= PPPlace_R1_L3_S2_NP5
FDAT_ACT= FPlace_R1_L3_S2_NP5
BAS(#PTP_PARAMS,100)
PTP XPlace_R1_L3_S2_NP5 C_DIS
;ENDFOLD
TRIGGER WHEN DISTANCE=1 DELAY=-1 DO Schrittmerker_R1Place(10203,10204,FPlace_R1_L3_S2_NP6,XPlace_R1_L3_S2_NP6) PRIO=-1
;FOLD PTP Place_R1_L3_S2_NP6 CONT Vel=100 % PPlace_R1_L3_S2_NP6 Tool[2]:Lower Gripper Base[0];%{PE}%R8.3.21,%MKUKATPBASIS,%CMOVE,%VPTP,%P 1:PTP, 2:Place_R1_L3_S2_NP6, 3:C_DIS, 5:100, 7:PPlace_R1_L3_S2_NP6
$BWDSTART=FALSE
PDAT_ACT= PPPlace_R1_L3_S2_NP6
FDAT_ACT= FPlace_R1_L3_S2_NP6
BAS(#PTP_PARAMS,100)
PTP XPlace_R1_L3_S2_NP6 C_DIS
;ENDFOLD

TRIGGER WHEN DISTANCE=1 DELAY=-1 DO Schrittmerker_R1Place(10204,10002,FHOME1,$nullframe,XHOME1) PRIO=-1
;FOLD PTP HOME1 Vel=100 % PHome1;%{PE}%R8.3.21,%MKUKATPBASIS,%CMOVE,%VPTP,%P 1:PTP, 2:HOME1, 3:, 5:100, 7:PHome1
$BWDSTART=FALSE
PDAT_ACT= PPHome1
FDAT_ACT= FHOME1
BAS(#PTP_PARAMS,100)
PTP XHOME1
;ENDFOLD

;***************************************************
;FOLD Final tasks.
; Robot out of area Rack 1 Level 3
RobAusStorage1_3_A69=RESET_IN_AREA
;***************************************************
; stop cyclic clearence check
$CYCFLAG[ciFreigabeSPS]=DISABLE_MONITORING
;***************************************************
; Disable collision detection
;FOLD COLLDETECT Off ;%{PE}
;FOLD Parameters ;%{h}
;Params IlfProvider=kukaroboter.basistech.inlineforms.colldetect.off; CollDetect.Command=Off
;ENDFOLD
USE_CD_PARAMS(0)
;ENDFOLD
;***************************************************
;ENDFOLD
;***************************************************

END

; ##################################################

GLOBAL DEF UP_Place_R1_L3_S3( )
;***************************************************
; Place part on:
;    Rack  1
;    Level 3
;    Shelf 3
;***************************************************
;FOLD Preconditions - Vorraussetzungen
;***************************************************
; Enable collision detection
;FOLD COLLDETECT SetLimits Axis1: 150 % Axis2: 200 % Axis3: 150 % Axis4: 200 % Axis5: 150 % Axis6: 150 % ;%{PE}
;FOLD Parameters ;%{h}
;Params IlfProvider=kukaroboter.basistech.inlineforms.colldetect.setlimits; CollDetect.Command=SetLimits; CollDetect.Axis1=150; CollDetect.Axis2=200; CollDetect.Axis3=150; CollDetect.Axis4=200; CollDetect.Axis5=150; CollDetect.Axis6=150
;ENDFOLD
SET_TQ_VALUES(150, 200, 150, 200, 150, 150)
;ENDFOLD
;***************************************************
; Check for part in gripper (tool 2).
CheckPartPresent(OCCUPIED_GRIPPER,PART_ON_TOOL_2)
;***************************************************
; Enable part lost detection for tool 2
SetPartLostDetection(PART_ON_TOOL_2)
;***************************************************
; Set load data.
SetLoadData( )
;***************************************************
; Robot has to start from home position.
IF NOT $IN_HOME1 THEN
  UP_HomeToHome(1)
ENDIF
;***************************************************
;ENDFOLD

TRIGGER WHEN DISTANCE=1 DELAY=-1 DO Schrittmerker_R1Place(10002,10002,FHOME1,$nullframe,XHOME1) PRIO=-1
;FOLD PTP HOME1 Vel=12 % PHome1;%{PE}%R8.3.21,%MKUKATPBASIS,%CMOVE,%VPTP,%P 1:PTP, 2:HOME1, 3:, 5:12, 7:PHome1
$BWDSTART=FALSE
PDAT_ACT= PPHome1
FDAT_ACT= FHOME1
BAS(#PTP_PARAMS,12)
PTP XHOME1
;ENDFOLD

;***************************************************
;FOLD Area clearence handshake.
IF NOT $FLAG[M_Inbetriebnahme] THEN
  ;-------------------------------------------------
  ; Request area clearence.
  AnfStoer_Store1_3_A101=SET_REQUEST
  ;-------------------------------------------------
  ; Wait for area clearence from PLC.
  WAIT_FOR_INPUT("Frg_Storage1_3_E69",TRUE)
  ;-------------------------------------------------
  ; Reset area clearence request.
  AnfStoer_Store1_3_A101=RESET_REQUEST
  ;-------------------------------------------------
  ; start cyclic clearence check
  $CYCFLAG[ciFreigabeSPS]=Frg_Storage1_3_E69
  ;-------------------------------------------------
ENDIF
;***************************************************
; set "robot in area"
RobAusStorage1_3_A69=SET_IN_AREA
;ENDFOLD
;***************************************************

;***************************************************
;FOLD Check for Teachmode
IF $FLAG[M_Teachen] THEN
  WAIT FOR $T1
ENDIF
;ENDFOLD
;***************************************************

; move to the rack
TRIGGER WHEN DISTANCE=1 DELAY=-1 DO Schrittmerker_R1Place(10210,10002,FPlace_R1_L3_S3_VP1,XPlace_R1_L3_S3_VP1) PRIO=-1
;FOLD PTP Place_R1_L3_S3_VP1 CONT Vel=12 % PPlace_R1_L3_S3_VP1 Tool[2]:Lower Gripper Base[0];%{PE}%R8.3.21,%MKUKATPBASIS,%CMOVE,%VPTP,%P 1:PTP, 2:Place_R1_L3_S3_VP1, 3:C_DIS, 5:12, 7:PPlace_R1_L3_S3_VP1
$BWDSTART=FALSE
PDAT_ACT= PPPlace_R1_L3_S3_VP1
FDAT_ACT= FPlace_R1_L3_S3_VP1
BAS(#PTP_PARAMS,12)
PTP XPlace_R1_L3_S3_VP1 C_DIS
;ENDFOLD
TRIGGER WHEN DISTANCE=1 DELAY=-1 DO Schrittmerker_R1Place(10211,10210,FPlace_R1_L3_S3_VP2,XPlace_R1_L3_S3_VP2) PRIO=-1
;FOLD PTP Place_R1_L3_S3_VP2 CONT Vel=12 % PPlace_R1_L3_S3_VP2 Tool[2]:Lower Gripper Base[0];%{PE}%R8.3.21,%MKUKATPBASIS,%CMOVE,%VPTP,%P 1:PTP, 2:Place_R1_L3_S3_VP2, 3:C_DIS, 5:12, 7:PPlace_R1_L3_S3_VP2
$BWDSTART=FALSE
PDAT_ACT= PPPlace_R1_L3_S3_VP2
FDAT_ACT= FPlace_R1_L3_S3_VP2
BAS(#PTP_PARAMS,12)
PTP XPlace_R1_L3_S3_VP2 C_DIS
;ENDFOLD
TRIGGER WHEN DISTANCE=1 DELAY=-1 DO Schrittmerker_R1Place(10212,10211,FPlace_R1_L3_S3_VP3,XPlace_R1_L3_S3_VP3) PRIO=-1
;FOLD PTP Place_R1_L3_S3_VP3 CONT Vel=12 % PPlace_R1_L3_S3_VP3 Tool[2]:Lower Gripper Base[0];%{PE}%R8.3.21,%MKUKATPBASIS,%CMOVE,%VPTP,%P 1:PTP, 2:Place_R1_L3_S3_VP3, 3:C_DIS, 5:12, 7:PPlace_R1_L3_S3_VP3
$BWDSTART=FALSE
PDAT_ACT= PPPlace_R1_L3_S3_VP3
FDAT_ACT= FPlace_R1_L3_S3_VP3
BAS(#PTP_PARAMS,12)
PTP XPlace_R1_L3_S3_VP3 C_DIS
;ENDFOLD
TRIGGER WHEN DISTANCE=1 DELAY=-1 DO Schrittmerker_R1Place(10213,10212,FPlace_R1_L3_S3_VP4,XPlace_R1_L3_S3_VP4) PRIO=-1
;FOLD PTP Place_R1_L3_S3_VP4 CONT Vel=12 % PPlace_R1_L3_S3_VP4 Tool[2]:Lower Gripper Base[0];%{PE}%R8.3.21,%MKUKATPBASIS,%CMOVE,%VPTP,%P 1:PTP, 2:Place_R1_L3_S3_VP4, 3:C_DIS, 5:12, 7:PPlace_R1_L3_S3_VP4
$BWDSTART=FALSE
PDAT_ACT= PPPlace_R1_L3_S3_VP4
FDAT_ACT= FPlace_R1_L3_S3_VP4
BAS(#PTP_PARAMS,12)
PTP XPlace_R1_L3_S3_VP4 C_DIS
;ENDFOLD
TRIGGER WHEN DISTANCE=1 DELAY=-1 DO Schrittmerker_R1Place(10214,10213,FPlace_R1_L3_S3_VP5,XPlace_R1_L3_S3_VP5) PRIO=-1
;FOLD PTP Place_R1_L3_S3_VP5 CONT Vel=12 % PPlace_R1_L3_S3_VP5 Tool[2]:Lower Gripper Base[1]:Rack1;%{PE}%R8.3.21,%MKUKATPBASIS,%CMOVE,%VPTP,%P 1:PTP, 2:Place_R1_L3_S3_VP5, 3:C_DIS, 5:12, 7:PPlace_R1_L3_S3_VP5
$BWDSTART=FALSE
PDAT_ACT= PPPlace_R1_L3_S3_VP5
FDAT_ACT= FPlace_R1_L3_S3_VP5
BAS(#PTP_PARAMS,12)
PTP XPlace_R1_L3_S3_VP5 C_DIS
;ENDFOLD

TRIGGER WHEN DISTANCE=1 DELAY=-1 DO Schrittmerker_R1Place(10215,10214,FPlace_R1_L3_S3_Check,XPlace_R1_L3_S3_Check) PRIO=-1
;FOLD PTP Place_R1_L3_S3_Check Vel=12 % PPlace_R1_L3_S3_Check Tool[2]:Lower Gripper Base[1]:Rack1;%{PE}%R8.3.21,%MKUKATPBASIS,%CMOVE,%VPTP,%P 1:PTP, 2:Place_R1_L3_S3_Check, 3:, 5:12, 7:PPlace_R1_L3_S3_Check
$BWDSTART=FALSE
PDAT_ACT= PPPlace_R1_L3_S3_Check
FDAT_ACT= FPlace_R1_L3_S3_Check
BAS(#PTP_PARAMS,12)
PTP XPlace_R1_L3_S3_Check
;ENDFOLD

;***************************************************
;FOLD Pruefe Platz frei
IF (DetectPart(CHECK_SHELF,PLACE)==OCCUPIED) THEN
  UP_Rueckzug_R1Place( )
  RETURN
ENDIF
;ENDFOLD
;***************************************************

TRIGGER WHEN DISTANCE=1 DELAY=-1 DO Schrittmerker_R1Place(10216,10215,FPlace_R1_L3_S3_VP6,XPlace_R1_L3_S3_VP6) PRIO=-1
;FOLD LIN Place_R1_L3_S3_VP6 CONT Vel=0.5 m/s LPlace_R1_L3_S3_VP6 Tool[2]:Lower Gripper Base[1]:Rack1;%{PE}%R8.3.21,%MKUKATPBASIS,%CMOVE,%VLIN,%P 1:LIN, 2:Place_R1_L3_S3_VP6, 3:C_DIS C_DIS, 5:0.5, 7:LPlace_R1_L3_S3_VP6
$BWDSTART=FALSE
LDAT_ACT= LLPlace_R1_L3_S3_VP6
FDAT_ACT= FPlace_R1_L3_S3_VP6
BAS(#CP_PARAMS,0.5)
LIN XPlace_R1_L3_S3_VP6 C_DIS C_DIS
;ENDFOLD
TRIGGER WHEN DISTANCE=1 DELAY=-1 DO Schrittmerker_R1Place(10217,10216,FPlace_R1_L3_S3_VP7,XPlace_R1_L3_S3_VP7) PRIO=-1
;FOLD LIN Place_R1_L3_S3_VP7 CONT Vel=0.5 m/s LPlace_R1_L3_S3_VP7 Tool[2]:Lower Gripper Base[1]:Rack1;%{PE}%R8.3.21,%MKUKATPBASIS,%CMOVE,%VLIN,%P 1:LIN, 2:Place_R1_L3_S3_VP7, 3:C_DIS C_DIS, 5:0.5, 7:LPlace_R1_L3_S3_VP7
$BWDSTART=FALSE
LDAT_ACT= LLPlace_R1_L3_S3_VP7
FDAT_ACT= FPlace_R1_L3_S3_VP7
BAS(#CP_PARAMS,0.5)
LIN XPlace_R1_L3_S3_VP7 C_DIS C_DIS
;ENDFOLD

;FOLD Test the way back home - part 1
CONTINUE
IF ($FLAG[M_Test_GrdstFahren1] AND NOT $FLAG[M_Test_GrdstFahren2]) THEN
  $FLAG[M_Test_GrdstFahren2]=TRUE
  UP_Rueckzug( )
  RETURN
ENDIF
;ENDFOLD

;-------------------------------
; Place part position
;-------------------------------
TRIGGER WHEN DISTANCE=1 DELAY=-1 DO Schrittmerker_R1Place(10218,10219,FPlace_R1_L3_S3_AP,XPlace_R1_L3_S3_AP) PRIO=-1
;FOLD LIN Place_R1_L3_S3_AP Vel=0.2 m/s LPlace_R1_L3_S3_AP Tool[2]:Lower Gripper Base[1]:Rack1;%{PE}%R8.3.21,%MKUKATPBASIS,%CMOVE,%VLIN,%P 1:LIN, 2:Place_R1_L3_S3_AP, 3:, 5:0.2, 7:LPlace_R1_L3_S3_AP
$BWDSTART=FALSE
LDAT_ACT= LLPlace_R1_L3_S3_AP
FDAT_ACT= FPlace_R1_L3_S3_AP
BAS(#CP_PARAMS,0.2)
LIN XPlace_R1_L3_S3_AP
;ENDFOLD

;FOLD Test the way back home - part 2
CONTINUE
IF $FLAG[M_Test_GrdstFahren2] THEN
  $FLAG[M_Test_GrdstFahren2]=FALSE
  UP_Rueckzug( )
  RETURN
ENDIF
;ENDFOLD

;***************************************************
; Disable part lost detection
SetPartLostDetection(NO_PART)
;***************************************************

TRIGGER WHEN DISTANCE=1 DELAY=-1 DO Schrittmerker_R1Place(10219,10220,FPlace_R1_L3_S3_NP1,XPlace_R1_L3_S3_NP1) PRIO=-1
;FOLD LIN Place_R1_L3_S3_NP1 Vel=0.2 m/s LPlace_R1_L3_S3_NP1 Tool[2]:Lower Gripper Base[1]:Rack1;%{PE}%R8.3.21,%MKUKATPBASIS,%CMOVE,%VLIN,%P 1:LIN, 2:Place_R1_L3_S3_NP1, 3:C_DIS C_DIS, 5:0.2, 7:LPlace_R1_L3_S3_NP1
$BWDSTART=FALSE
LDAT_ACT= LLPlace_R1_L3_S3_NP1
FDAT_ACT= FPlace_R1_L3_S3_NP1
BAS(#CP_PARAMS,0.2)
LIN XPlace_R1_L3_S3_NP1
;ENDFOLD

;***************************************************
; Check for part present (empty gripper)
CheckPartPresent(EMPTY_GRIPPER)
;***************************************************
; set load data
SetLoadData( )
;***************************************************

TRIGGER WHEN DISTANCE=1 DELAY=-1 DO Schrittmerker_R1Place(10220,10221,FPlace_R1_L3_S3_NP2,XPlace_R1_L3_S3_NP2) PRIO=-1
;FOLD LIN Place_R1_L3_S3_NP2 Vel=0.5 m/s LPlace_R1_L3_S3_NP2 Tool[2]:Lower Gripper Base[1]:Rack1;%{PE}%R8.3.21,%MKUKATPBASIS,%CMOVE,%VLIN,%P 1:LIN, 2:Place_R1_L3_S3_NP2, 3:, 5:0.5, 7:LPlace_R1_L3_S3_NP2
$BWDSTART=FALSE
LDAT_ACT= LLPlace_R1_L3_S3_NP2
FDAT_ACT= FPlace_R1_L3_S3_NP2
BAS(#CP_PARAMS,0.5)
LIN XPlace_R1_L3_S3_NP2
;ENDFOLD
TRIGGER WHEN DISTANCE=1 DELAY=-1 DO Schrittmerker_R1Place(10221,10222,FPlace_R1_L3_S3_NP3,XPlace_R1_L3_S3_NP3) PRIO=-1
;FOLD PTP Place_R1_L3_S3_NP3 CONT Vel=100 % PPlace_R1_L3_S3_NP3 Tool[2]:Lower Gripper Base[0];%{PE}%R8.3.21,%MKUKATPBASIS,%CMOVE,%VPTP,%P 1:PTP, 2:Place_R1_L3_S3_NP3, 3:C_DIS, 5:100, 7:PPlace_R1_L3_S3_NP3
$BWDSTART=FALSE
PDAT_ACT= PPPlace_R1_L3_S3_NP3
FDAT_ACT= FPlace_R1_L3_S3_NP3
BAS(#PTP_PARAMS,100)
PTP XPlace_R1_L3_S3_NP3 C_DIS
;ENDFOLD
TRIGGER WHEN DISTANCE=1 DELAY=-1 DO Schrittmerker_R1Place(10222,10223,FPlace_R1_L3_S3_NP4,XPlace_R1_L3_S3_NP4) PRIO=-1
;FOLD PTP Place_R1_L3_S3_NP4 CONT Vel=100 % PPlace_R1_L3_S3_NP4 Tool[2]:Lower Gripper Base[0];%{PE}%R8.3.21,%MKUKATPBASIS,%CMOVE,%VPTP,%P 1:PTP, 2:Place_R1_L3_S3_NP4, 3:C_DIS, 5:100, 7:PPlace_R1_L3_S3_NP4
$BWDSTART=FALSE
PDAT_ACT= PPPlace_R1_L3_S3_NP4
FDAT_ACT= FPlace_R1_L3_S3_NP4
BAS(#PTP_PARAMS,100)
PTP XPlace_R1_L3_S3_NP4 C_DIS
;ENDFOLD
TRIGGER WHEN DISTANCE=1 DELAY=-1 DO Schrittmerker_R1Place(10223,10224,FPlace_R1_L3_S3_NP5,XPlace_R1_L3_S3_NP5) PRIO=-1
;FOLD PTP Place_R1_L3_S3_NP5 CONT Vel=100 % PPlace_R1_L3_S3_NP5 Tool[2]:Lower Gripper Base[0];%{PE}%R8.3.21,%MKUKATPBASIS,%CMOVE,%VPTP,%P 1:PTP, 2:Place_R1_L3_S3_NP5, 3:C_DIS, 5:100, 7:PPlace_R1_L3_S3_NP5
$BWDSTART=FALSE
PDAT_ACT= PPPlace_R1_L3_S3_NP5
FDAT_ACT= FPlace_R1_L3_S3_NP5
BAS(#PTP_PARAMS,100)
PTP XPlace_R1_L3_S3_NP5 C_DIS
;ENDFOLD
TRIGGER WHEN DISTANCE=1 DELAY=-1 DO Schrittmerker_R1Place(10224,10225,FPlace_R1_L3_S3_NP6,XPlace_R1_L3_S3_NP6) PRIO=-1
;FOLD PTP Place_R1_L3_S3_NP6 CONT Vel=100 % PPlace_R1_L3_S3_NP6 Tool[2]:Lower Gripper Base[0];%{PE}%R8.3.21,%MKUKATPBASIS,%CMOVE,%VPTP,%P 1:PTP, 2:Place_R1_L3_S3_NP6, 3:C_DIS, 5:100, 7:PPlace_R1_L3_S3_NP6
$BWDSTART=FALSE
PDAT_ACT= PPPlace_R1_L3_S3_NP6
FDAT_ACT= FPlace_R1_L3_S3_NP6
BAS(#PTP_PARAMS,100)
PTP XPlace_R1_L3_S3_NP6 C_DIS
;ENDFOLD
TRIGGER WHEN DISTANCE=1 DELAY=-1 DO Schrittmerker_R1Place(10225,10226,FPlace_R1_L3_S3_NP7,XPlace_R1_L3_S3_NP7) PRIO=-1
;FOLD PTP Place_R1_L3_S3_NP7 CONT Vel=100 % PPlace_R1_L3_S3_NP7 Tool[2]:Lower Gripper Base[0];%{PE}%R8.3.21,%MKUKATPBASIS,%CMOVE,%VPTP,%P 1:PTP, 2:Place_R1_L3_S3_NP7, 3:C_DIS, 5:100, 7:PPlace_R1_L3_S3_NP7
$BWDSTART=FALSE
PDAT_ACT= PPPlace_R1_L3_S3_NP7
FDAT_ACT= FPlace_R1_L3_S3_NP7
BAS(#PTP_PARAMS,100)
PTP XPlace_R1_L3_S3_NP7 C_DIS
;ENDFOLD

TRIGGER WHEN DISTANCE=1 DELAY=-1 DO Schrittmerker_R1Place(10226,10002,FHOME1,$nullframe,XHOME1) PRIO=-1
;FOLD PTP HOME1 Vel=100 % PHome1;%{PE}%R8.3.21,%MKUKATPBASIS,%CMOVE,%VPTP,%P 1:PTP, 2:HOME1, 3:, 5:100, 7:PHome1
$BWDSTART=FALSE
PDAT_ACT= PPHome1
FDAT_ACT= FHOME1
BAS(#PTP_PARAMS,100)
PTP XHOME1
;ENDFOLD

;***************************************************
;FOLD Final tasks.
; Robot out of area Rack 1 Level 3
RobAusStorage1_3_A69=RESET_IN_AREA
;***************************************************
; stop cyclic clearence check
$CYCFLAG[ciFreigabeSPS]=DISABLE_MONITORING
;***************************************************
; Disable collision detection
;FOLD COLLDETECT Off ;%{PE}
;FOLD Parameters ;%{h}
;Params IlfProvider=kukaroboter.basistech.inlineforms.colldetect.off; CollDetect.Command=Off
;ENDFOLD
USE_CD_PARAMS(0)
;ENDFOLD
;***************************************************
;ENDFOLD
;***************************************************

END

; ##################################################

GLOBAL DEF UP_Place_R1_L3_S4( )
;***************************************************
; Place part on:
;    Rack  1
;    Level 3
;    Shelf 4
;***************************************************
;FOLD Preconditions - Vorraussetzungen
;***************************************************
; Enable collision detection
;FOLD COLLDETECT SetLimits Axis1: 150 % Axis2: 200 % Axis3: 150 % Axis4: 200 % Axis5: 150 % Axis6: 150 % ;%{PE}
;FOLD Parameters ;%{h}
;Params IlfProvider=kukaroboter.basistech.inlineforms.colldetect.setlimits; CollDetect.Command=SetLimits; CollDetect.Axis1=150; CollDetect.Axis2=200; CollDetect.Axis3=150; CollDetect.Axis4=200; CollDetect.Axis5=150; CollDetect.Axis6=150
;ENDFOLD
SET_TQ_VALUES(150, 200, 150, 200, 150, 150)
;ENDFOLD
;***************************************************
; Check for part in gripper (tool 2).
CheckPartPresent(OCCUPIED_GRIPPER,PART_ON_TOOL_2)
;***************************************************
; Enable part lost detection for tool 2
SetPartLostDetection(PART_ON_TOOL_2)
;***************************************************
; Set load data.
SetLoadData( )
;***************************************************
; Robot has to start from home position.
IF NOT $IN_HOME1 THEN
  UP_HomeToHome(1)
ENDIF
;***************************************************
;ENDFOLD

TRIGGER WHEN DISTANCE=1 DELAY=-1 DO Schrittmerker_R1Place(10002,10002,FHOME1,$nullframe,XHOME1) PRIO=-1
;FOLD PTP HOME1 Vel=12 % PHome1;%{PE}%R8.3.21,%MKUKATPBASIS,%CMOVE,%VPTP,%P 1:PTP, 2:HOME1, 3:, 5:12, 7:PHome1
$BWDSTART=FALSE
PDAT_ACT= PPHome1
FDAT_ACT= FHOME1
BAS(#PTP_PARAMS,12)
PTP XHOME1
;ENDFOLD

;***************************************************
;FOLD Area clearence handshake.
IF NOT $FLAG[M_Inbetriebnahme] THEN
  ;-------------------------------------------------
  ; Request area clearence.
  AnfStoer_Store1_3_A101=SET_REQUEST
  ;-------------------------------------------------
  ; Wait for area clearence from PLC.
  WAIT_FOR_INPUT("Frg_Storage1_3_E69",TRUE)
  ;-------------------------------------------------
  ; Reset area clearence request.
  AnfStoer_Store1_3_A101=RESET_REQUEST
  ;-------------------------------------------------
  ; start cyclic clearence check
  $CYCFLAG[ciFreigabeSPS]=Frg_Storage1_3_E69
  ;-------------------------------------------------
ENDIF
;***************************************************
; set "robot in area"
RobAusStorage1_3_A69=SET_IN_AREA
;ENDFOLD
;***************************************************

;***************************************************
;FOLD Check for Teachmode
IF $FLAG[M_Teachen] THEN
  WAIT FOR $T1
ENDIF
;ENDFOLD
;***************************************************

; move to the rack
TRIGGER WHEN DISTANCE=1 DELAY=-1 DO Schrittmerker_R1Place(10230,10002,FPlace_R1_L3_S4_VP1,XPlace_R1_L3_S4_VP1) PRIO=-1
;FOLD PTP Place_R1_L3_S4_VP1 CONT Vel=12 % PPlace_R1_L3_S4_VP1 Tool[2]:Lower Gripper Base[0];%{PE}%R8.3.21,%MKUKATPBASIS,%CMOVE,%VPTP,%P 1:PTP, 2:Place_R1_L3_S4_VP1, 3:C_DIS, 5:12, 7:PPlace_R1_L3_S4_VP1
$BWDSTART=FALSE
PDAT_ACT= PPPlace_R1_L3_S4_VP1
FDAT_ACT= FPlace_R1_L3_S4_VP1
BAS(#PTP_PARAMS,12)
PTP XPlace_R1_L3_S4_VP1 C_DIS
;ENDFOLD
TRIGGER WHEN DISTANCE=1 DELAY=-1 DO Schrittmerker_R1Place(10231,10230,FPlace_R1_L3_S4_VP2,XPlace_R1_L3_S4_VP2) PRIO=-1
;FOLD PTP Place_R1_L3_S4_VP2 CONT Vel=12 % PPlace_R1_L3_S4_VP2 Tool[2]:Lower Gripper Base[0];%{PE}%R8.3.21,%MKUKATPBASIS,%CMOVE,%VPTP,%P 1:PTP, 2:Place_R1_L3_S4_VP2, 3:C_DIS, 5:12, 7:PPlace_R1_L3_S4_VP2
$BWDSTART=FALSE
PDAT_ACT= PPPlace_R1_L3_S4_VP2
FDAT_ACT= FPlace_R1_L3_S4_VP2
BAS(#PTP_PARAMS,12)
PTP XPlace_R1_L3_S4_VP2 C_DIS
;ENDFOLD
TRIGGER WHEN DISTANCE=1 DELAY=-1 DO Schrittmerker_R1Place(10232,10231,FPlace_R1_L3_S4_VP3,XPlace_R1_L3_S4_VP3) PRIO=-1
;FOLD PTP Place_R1_L3_S4_VP3 CONT Vel=12 % PPlace_R1_L3_S4_VP3 Tool[2]:Lower Gripper Base[0];%{PE}%R8.3.21,%MKUKATPBASIS,%CMOVE,%VPTP,%P 1:PTP, 2:Place_R1_L3_S4_VP3, 3:C_DIS, 5:12, 7:PPlace_R1_L3_S4_VP3
$BWDSTART=FALSE
PDAT_ACT= PPPlace_R1_L3_S4_VP3
FDAT_ACT= FPlace_R1_L3_S4_VP3
BAS(#PTP_PARAMS,12)
PTP XPlace_R1_L3_S4_VP3 C_DIS
;ENDFOLD
TRIGGER WHEN DISTANCE=1 DELAY=-1 DO Schrittmerker_R1Place(10233,10232,FPlace_R1_L3_S4_VP4,XPlace_R1_L3_S4_VP4) PRIO=-1
;FOLD PTP Place_R1_L3_S4_VP4 CONT Vel=12 % PPlace_R1_L3_S4_VP4 Tool[2]:Lower Gripper Base[0];%{PE}%R8.3.21,%MKUKATPBASIS,%CMOVE,%VPTP,%P 1:PTP, 2:Place_R1_L3_S4_VP4, 3:C_DIS, 5:12, 7:PPlace_R1_L3_S4_VP4
$BWDSTART=FALSE
PDAT_ACT= PPPlace_R1_L3_S4_VP4
FDAT_ACT= FPlace_R1_L3_S4_VP4
BAS(#PTP_PARAMS,12)
PTP XPlace_R1_L3_S4_VP4 C_DIS
;ENDFOLD
TRIGGER WHEN DISTANCE=1 DELAY=-1 DO Schrittmerker_R1Place(10234,10233,FPlace_R1_L3_S4_VP5,XPlace_R1_L3_S4_VP5) PRIO=-1
;FOLD PTP Place_R1_L3_S4_VP5 CONT Vel=12 % PPlace_R1_L3_S4_VP5 Tool[2]:Lower Gripper Base[1]:Rack1;%{PE}%R8.3.21,%MKUKATPBASIS,%CMOVE,%VPTP,%P 1:PTP, 2:Place_R1_L3_S4_VP5, 3:C_DIS, 5:12, 7:PPlace_R1_L3_S4_VP5
$BWDSTART=FALSE
PDAT_ACT= PPPlace_R1_L3_S4_VP5
FDAT_ACT= FPlace_R1_L3_S4_VP5
BAS(#PTP_PARAMS,12)
PTP XPlace_R1_L3_S4_VP5 C_DIS
;ENDFOLD

TRIGGER WHEN DISTANCE=1 DELAY=-1 DO Schrittmerker_R1Place(10235,10234,FPlace_R1_L3_S4_Check,XPlace_R1_L3_S4_Check) PRIO=-1
;FOLD PTP Place_R1_L3_S4_Check Vel=12 % PPlace_R1_L3_S4_Check Tool[2]:Lower Gripper Base[1]:Rack1;%{PE}%R8.3.21,%MKUKATPBASIS,%CMOVE,%VPTP,%P 1:PTP, 2:Place_R1_L3_S4_Check, 3:, 5:12, 7:PPlace_R1_L3_S4_Check
$BWDSTART=FALSE
PDAT_ACT= PPPlace_R1_L3_S4_Check
FDAT_ACT= FPlace_R1_L3_S4_Check
BAS(#PTP_PARAMS,12)
PTP XPlace_R1_L3_S4_Check
;ENDFOLD

;***************************************************
;FOLD Pruefe Platz frei
IF (DetectPart(CHECK_SHELF,PLACE)==OCCUPIED) THEN
  UP_Rueckzug_R1Place( )
  RETURN
ENDIF
;ENDFOLD
;***************************************************

TRIGGER WHEN DISTANCE=1 DELAY=-1 DO Schrittmerker_R1Place(10236,10235,FPlace_R1_L3_S4_VP6,XPlace_R1_L3_S4_VP6) PRIO=-1
;FOLD LIN Place_R1_L3_S4_VP6 CONT Vel=0.5 m/s LPlace_R1_L3_S4_VP6 Tool[2]:Lower Gripper Base[1]:Rack1;%{PE}%R8.3.21,%MKUKATPBASIS,%CMOVE,%VLIN,%P 1:LIN, 2:Place_R1_L3_S4_VP6, 3:C_DIS C_DIS, 5:0.5, 7:LPlace_R1_L3_S4_VP6
$BWDSTART=FALSE
LDAT_ACT= LLPlace_R1_L3_S4_VP6
FDAT_ACT= FPlace_R1_L3_S4_VP6
BAS(#CP_PARAMS,0.5)
LIN XPlace_R1_L3_S4_VP6 C_DIS C_DIS
;ENDFOLD
TRIGGER WHEN DISTANCE=1 DELAY=-1 DO Schrittmerker_R1Place(10237,10236,FPlace_R1_L3_S4_VP7,XPlace_R1_L3_S4_VP7) PRIO=-1
;FOLD LIN Place_R1_L3_S4_VP7 CONT Vel=0.5 m/s LPlace_R1_L3_S4_VP7 Tool[2]:Lower Gripper Base[1]:Rack1;%{PE}%R8.3.21,%MKUKATPBASIS,%CMOVE,%VLIN,%P 1:LIN, 2:Place_R1_L3_S4_VP7, 3:C_DIS C_DIS, 5:0.5, 7:LPlace_R1_L3_S4_VP7
$BWDSTART=FALSE
LDAT_ACT= LLPlace_R1_L3_S4_VP7
FDAT_ACT= FPlace_R1_L3_S4_VP7
BAS(#CP_PARAMS,0.5)
LIN XPlace_R1_L3_S4_VP7 C_DIS C_DIS
;ENDFOLD

;FOLD Test the way back home - part 1
CONTINUE
IF ($FLAG[M_Test_GrdstFahren1] AND NOT $FLAG[M_Test_GrdstFahren2]) THEN
  $FLAG[M_Test_GrdstFahren2]=TRUE
  UP_Rueckzug( )
  RETURN
ENDIF
;ENDFOLD

;-------------------------------
; Place part position
;-------------------------------
TRIGGER WHEN DISTANCE=1 DELAY=-1 DO Schrittmerker_R1Place(10238,10239,FPlace_R1_L3_S4_AP,XPlace_R1_L3_S4_AP) PRIO=-1
;FOLD LIN Place_R1_L3_S4_AP Vel=0.2 m/s LPlace_R1_L3_S4_AP Tool[2]:Lower Gripper Base[1]:Rack1;%{PE}%R8.3.21,%MKUKATPBASIS,%CMOVE,%VLIN,%P 1:LIN, 2:Place_R1_L3_S4_AP, 3:, 5:0.2, 7:LPlace_R1_L3_S4_AP
$BWDSTART=FALSE
LDAT_ACT= LLPlace_R1_L3_S4_AP
FDAT_ACT= FPlace_R1_L3_S4_AP
BAS(#CP_PARAMS,0.2)
LIN XPlace_R1_L3_S4_AP
;ENDFOLD

;FOLD Test the way back home - part 2
CONTINUE
IF $FLAG[M_Test_GrdstFahren2] THEN
  $FLAG[M_Test_GrdstFahren2]=FALSE
  UP_Rueckzug( )
  RETURN
ENDIF
;ENDFOLD

;***************************************************
; Disable part lost detection
SetPartLostDetection(NO_PART)
;***************************************************

TRIGGER WHEN DISTANCE=1 DELAY=-1 DO Schrittmerker_R1Place(10239,10240,FPlace_R1_L3_S4_NP1,XPlace_R1_L3_S4_NP1) PRIO=-1
;FOLD LIN Place_R1_L3_S4_NP1 Vel=0.2 m/s LPlace_R1_L3_S4_NP1 Tool[2]:Lower Gripper Base[1]:Rack1;%{PE}%R8.3.21,%MKUKATPBASIS,%CMOVE,%VLIN,%P 1:LIN, 2:Place_R1_L3_S4_NP1, 3:C_DIS C_DIS, 5:0.2, 7:LPlace_R1_L3_S4_NP1
$BWDSTART=FALSE
LDAT_ACT= LLPlace_R1_L3_S4_NP1
FDAT_ACT= FPlace_R1_L3_S4_NP1
BAS(#CP_PARAMS,0.2)
LIN XPlace_R1_L3_S4_NP1
;ENDFOLD

;***************************************************
; Check for part present (empty gripper)
CheckPartPresent(EMPTY_GRIPPER)
;***************************************************
; set load data
SetLoadData( )
;***************************************************

TRIGGER WHEN DISTANCE=1 DELAY=-1 DO Schrittmerker_R1Place(10240,10241,FPlace_R1_L3_S4_NP2,XPlace_R1_L3_S4_NP2) PRIO=-1
;FOLD LIN Place_R1_L3_S4_NP2 CONT Vel=0.5 m/s LPlace_R1_L3_S4_NP2 Tool[2]:Lower Gripper Base[1]:Rack1;%{PE}%R8.3.21,%MKUKATPBASIS,%CMOVE,%VLIN,%P 1:LIN, 2:Place_R1_L3_S4_NP2, 3:C_DIS C_DIS, 5:0.5, 7:LPlace_R1_L3_S4_NP2
$BWDSTART=FALSE
LDAT_ACT= LLPlace_R1_L3_S4_NP2
FDAT_ACT= FPlace_R1_L3_S4_NP2
BAS(#CP_PARAMS,0.5)
LIN XPlace_R1_L3_S4_NP2 C_DIS C_DIS
;ENDFOLD
TRIGGER WHEN DISTANCE=1 DELAY=-1 DO Schrittmerker_R1Place(10241,10242,FPlace_R1_L3_S4_NP3,XPlace_R1_L3_S4_NP3) PRIO=-1
;FOLD LIN Place_R1_L3_S4_NP3 CONT Vel=0.5 m/s LPlace_R1_L3_S4_NP3 Tool[2]:Lower Gripper Base[1]:Rack1;%{PE}%R8.3.21,%MKUKATPBASIS,%CMOVE,%VLIN,%P 1:LIN, 2:Place_R1_L3_S4_NP3, 3:C_DIS C_DIS, 5:0.5, 7:LPlace_R1_L3_S4_NP3
$BWDSTART=FALSE
LDAT_ACT= LLPlace_R1_L3_S4_NP3
FDAT_ACT= FPlace_R1_L3_S4_NP3
BAS(#CP_PARAMS,0.5)
LIN XPlace_R1_L3_S4_NP3 C_DIS C_DIS
;ENDFOLD
TRIGGER WHEN DISTANCE=1 DELAY=-1 DO Schrittmerker_R1Place(10242,10243,FPlace_R1_L3_S4_NP4,XPlace_R1_L3_S4_NP4) PRIO=-1
;FOLD PTP Place_R1_L3_S4_NP4 CONT Vel=100 % PPlace_R1_L3_S4_NP4 Tool[2]:Lower Gripper Base[0];%{PE}%R8.3.21,%MKUKATPBASIS,%CMOVE,%VPTP,%P 1:PTP, 2:Place_R1_L3_S4_NP4, 3:C_DIS, 5:100, 7:PPlace_R1_L3_S4_NP4
$BWDSTART=FALSE
PDAT_ACT= PPPlace_R1_L3_S4_NP4
FDAT_ACT= FPlace_R1_L3_S4_NP4
BAS(#PTP_PARAMS,100)
PTP XPlace_R1_L3_S4_NP4 C_DIS
;ENDFOLD
TRIGGER WHEN DISTANCE=1 DELAY=-1 DO Schrittmerker_R1Place(10243,10244,FPlace_R1_L3_S4_NP5,XPlace_R1_L3_S4_NP5) PRIO=-1
;FOLD PTP Place_R1_L3_S4_NP5 CONT Vel=100 % PPlace_R1_L3_S4_NP5 Tool[2]:Lower Gripper Base[0];%{PE}%R8.3.21,%MKUKATPBASIS,%CMOVE,%VPTP,%P 1:PTP, 2:Place_R1_L3_S4_NP5, 3:C_DIS, 5:100, 7:PPlace_R1_L3_S4_NP5
$BWDSTART=FALSE
PDAT_ACT= PPPlace_R1_L3_S4_NP5
FDAT_ACT= FPlace_R1_L3_S4_NP5
BAS(#PTP_PARAMS,100)
PTP XPlace_R1_L3_S4_NP5 C_DIS
;ENDFOLD
TRIGGER WHEN DISTANCE=1 DELAY=-1 DO Schrittmerker_R1Place(10244,10245,FPlace_R1_L3_S4_NP6,XPlace_R1_L3_S4_NP6) PRIO=-1
;FOLD PTP Place_R1_L3_S4_NP6 CONT Vel=100 % PPlace_R1_L3_S4_NP6 Tool[2]:Lower Gripper Base[0];%{PE}%R8.3.21,%MKUKATPBASIS,%CMOVE,%VPTP,%P 1:PTP, 2:Place_R1_L3_S4_NP6, 3:C_DIS, 5:100, 7:PPlace_R1_L3_S4_NP6
$BWDSTART=FALSE
PDAT_ACT= PPPlace_R1_L3_S4_NP6
FDAT_ACT= FPlace_R1_L3_S4_NP6
BAS(#PTP_PARAMS,100)
PTP XPlace_R1_L3_S4_NP6 C_DIS
;ENDFOLD
TRIGGER WHEN DISTANCE=1 DELAY=-1 DO Schrittmerker_R1Place(10245,10246,FPlace_R1_L3_S4_NP7,XPlace_R1_L3_S4_NP7) PRIO=-1
;FOLD PTP Place_R1_L3_S4_NP7 CONT Vel=100 % PPlace_R1_L3_S4_NP7 Tool[2]:Lower Gripper Base[0];%{PE}%R8.3.21,%MKUKATPBASIS,%CMOVE,%VPTP,%P 1:PTP, 2:Place_R1_L3_S4_NP7, 3:C_DIS, 5:100, 7:PPlace_R1_L3_S4_NP7
$BWDSTART=FALSE
PDAT_ACT= PPPlace_R1_L3_S4_NP7
FDAT_ACT= FPlace_R1_L3_S4_NP7
BAS(#PTP_PARAMS,100)
PTP XPlace_R1_L3_S4_NP7 C_DIS
;ENDFOLD
TRIGGER WHEN DISTANCE=1 DELAY=-1 DO Schrittmerker_R1Place(10246,10247,FPlace_R1_L3_S4_NP8,XPlace_R1_L3_S4_NP8) PRIO=-1
;FOLD PTP Place_R1_L3_S4_NP8 CONT Vel=100 % PPlace_R1_L3_S4_NP8 Tool[2]:Lower Gripper Base[0];%{PE}%R8.3.21,%MKUKATPBASIS,%CMOVE,%VPTP,%P 1:PTP, 2:Place_R1_L3_S4_NP8, 3:C_DIS, 5:100, 7:PPlace_R1_L3_S4_NP8
$BWDSTART=FALSE
PDAT_ACT= PPPlace_R1_L3_S4_NP8
FDAT_ACT= FPlace_R1_L3_S4_NP8
BAS(#PTP_PARAMS,100)
PTP XPlace_R1_L3_S4_NP8 C_DIS
;ENDFOLD

TRIGGER WHEN DISTANCE=1 DELAY=-1 DO Schrittmerker_R1Place(10247,10002,FHOME1,$nullframe,XHOME1) PRIO=-1
;FOLD PTP HOME1 Vel=100 % PHome1;%{PE}%R8.3.21,%MKUKATPBASIS,%CMOVE,%VPTP,%P 1:PTP, 2:HOME1, 3:, 5:100, 7:PHome1
$BWDSTART=FALSE
PDAT_ACT= PPHome1
FDAT_ACT= FHOME1
BAS(#PTP_PARAMS,100)
PTP XHOME1
;ENDFOLD

;***************************************************
;FOLD Final tasks.
; Robot out of area Rack 1 Level 3
RobAusStorage1_3_A69=RESET_IN_AREA
;***************************************************
; stop cyclic clearence check
$CYCFLAG[ciFreigabeSPS]=DISABLE_MONITORING
;***************************************************
; Disable collision detection
;FOLD COLLDETECT Off ;%{PE}
;FOLD Parameters ;%{h}
;Params IlfProvider=kukaroboter.basistech.inlineforms.colldetect.off; CollDetect.Command=Off
;ENDFOLD
USE_CD_PARAMS(0)
;ENDFOLD
;***************************************************
;ENDFOLD
;***************************************************

END

; ##################################################

GLOBAL DEF UP_Place_R1_L4_S1( )
;***************************************************
; Place part on:
;    Rack  1
;    Level 4
;    Shelf 1
;***************************************************
;FOLD Preconditions - Vorraussetzungen
;***************************************************
; Enable collision detection
;FOLD COLLDETECT SetLimits Axis1: 150 % Axis2: 200 % Axis3: 150 % Axis4: 200 % Axis5: 150 % Axis6: 150 % ;%{PE}
;FOLD Parameters ;%{h}
;Params IlfProvider=kukaroboter.basistech.inlineforms.colldetect.setlimits; CollDetect.Command=SetLimits; CollDetect.Axis1=150; CollDetect.Axis2=200; CollDetect.Axis3=150; CollDetect.Axis4=200; CollDetect.Axis5=150; CollDetect.Axis6=150
;ENDFOLD
SET_TQ_VALUES(150, 200, 150, 200, 150, 150)
;ENDFOLD
;***************************************************
; Check for part in gripper (tool 2).
CheckPartPresent(OCCUPIED_GRIPPER,PART_ON_TOOL_2)
;***************************************************
; Enable part lost detection for tool 2
SetPartLostDetection(PART_ON_TOOL_2)
;***************************************************
; Set load data.
SetLoadData( )
;***************************************************
; Robot has to start from home position.
IF NOT $IN_HOME1 THEN
  UP_HomeToHome(1)
ENDIF
;***************************************************
;ENDFOLD

TRIGGER WHEN DISTANCE=1 DELAY=-1 DO Schrittmerker_R1Place(10002,10002,FHOME1,$nullframe,XHOME1) PRIO=-1
;FOLD PTP HOME1 Vel=12 % PHome1;%{PE}%R8.3.21,%MKUKATPBASIS,%CMOVE,%VPTP,%P 1:PTP, 2:HOME1, 3:, 5:12, 7:PHome1
$BWDSTART=FALSE
PDAT_ACT= PPHome1
FDAT_ACT= FHOME1
BAS(#PTP_PARAMS,12)
PTP XHOME1
;ENDFOLD

;***************************************************
;FOLD Area clearence handshake.
IF NOT $FLAG[M_Inbetriebnahme] THEN
  ;-------------------------------------------------
  ; Request area clearence.
  AnfStoer_Store1_4_A102=SET_REQUEST
  ;-------------------------------------------------
  ; Wait for area clearence from PLC.
  WAIT_FOR_INPUT("Frg_Storage1_4_E70",TRUE)
  ;-------------------------------------------------
  ; Reset area clearence request.
  AnfStoer_Store1_4_A102=RESET_REQUEST
  ;-------------------------------------------------
  ; start cyclic clearence check
  $CYCFLAG[ciFreigabeSPS]=Frg_Storage1_4_E70
  ;-------------------------------------------------
ENDIF
;***************************************************
; set "robot in area"
RobAusStorage1_4_A70=SET_IN_AREA
;ENDFOLD
;***************************************************

;***************************************************
;FOLD Check for Teachmode
IF $FLAG[M_Teachen] THEN
  WAIT FOR $T1
ENDIF
;ENDFOLD
;***************************************************

; move to the rack
TRIGGER WHEN DISTANCE=1 DELAY=-1 DO Schrittmerker_R1Place(10250,10002,FPlace_R1_L4_S1_VP1,XPlace_R1_L4_S1_VP1) PRIO=-1
;FOLD PTP Place_R1_L4_S1_VP1 CONT Vel=12 % PPlace_R1_L4_S1_VP1 Tool[2]:Lower Gripper Base[0];%{PE}%R8.3.21,%MKUKATPBASIS,%CMOVE,%VPTP,%P 1:PTP, 2:Place_R1_L4_S1_VP1, 3:C_DIS, 5:12, 7:PPlace_R1_L4_S1_VP1
$BWDSTART=FALSE
PDAT_ACT= PPPlace_R1_L4_S1_VP1
FDAT_ACT= FPlace_R1_L4_S1_VP1
BAS(#PTP_PARAMS,12)
PTP XPlace_R1_L4_S1_VP1 C_DIS
;ENDFOLD
TRIGGER WHEN DISTANCE=1 DELAY=-1 DO Schrittmerker_R1Place(10251,10250,FPlace_R1_L4_S1_VP2,XPlace_R1_L4_S1_VP2) PRIO=-1
;FOLD PTP Place_R1_L4_S1_VP2 CONT Vel=12 % PPlace_R1_L4_S1_VP2 Tool[2]:Lower Gripper Base[0];%{PE}%R8.3.21,%MKUKATPBASIS,%CMOVE,%VPTP,%P 1:PTP, 2:Place_R1_L4_S1_VP2, 3:C_DIS, 5:12, 7:PPlace_R1_L4_S1_VP2
$BWDSTART=FALSE
PDAT_ACT= PPPlace_R1_L4_S1_VP2
FDAT_ACT= FPlace_R1_L4_S1_VP2
BAS(#PTP_PARAMS,12)
PTP XPlace_R1_L4_S1_VP2 C_DIS
;ENDFOLD
TRIGGER WHEN DISTANCE=1 DELAY=-1 DO Schrittmerker_R1Place(10252,10251,FPlace_R1_L4_S1_VP3,XPlace_R1_L4_S1_VP3) PRIO=-1
;FOLD PTP Place_R1_L4_S1_VP3 CONT Vel=12 % PPlace_R1_L4_S1_VP3 Tool[2]:Lower Gripper Base[0];%{PE}%R8.3.21,%MKUKATPBASIS,%CMOVE,%VPTP,%P 1:PTP, 2:Place_R1_L4_S1_VP3, 3:C_DIS, 5:12, 7:PPlace_R1_L4_S1_VP3
$BWDSTART=FALSE
PDAT_ACT= PPPlace_R1_L4_S1_VP3
FDAT_ACT= FPlace_R1_L4_S1_VP3
BAS(#PTP_PARAMS,12)
PTP XPlace_R1_L4_S1_VP3 C_DIS
;ENDFOLD
TRIGGER WHEN DISTANCE=1 DELAY=-1 DO Schrittmerker_R1Place(10253,10252,FPlace_R1_L4_S1_VP4,XPlace_R1_L4_S1_VP4) PRIO=-1
;FOLD PTP Place_R1_L4_S1_VP4 CONT Vel=12 % PPlace_R1_L4_S1_VP4 Tool[2]:Lower Gripper Base[0];%{PE}%R8.3.21,%MKUKATPBASIS,%CMOVE,%VPTP,%P 1:PTP, 2:Place_R1_L4_S1_VP4, 3:C_DIS, 5:12, 7:PPlace_R1_L4_S1_VP4
$BWDSTART=FALSE
PDAT_ACT= PPPlace_R1_L4_S1_VP4
FDAT_ACT= FPlace_R1_L4_S1_VP4
BAS(#PTP_PARAMS,12)
PTP XPlace_R1_L4_S1_VP4 C_DIS
;ENDFOLD
TRIGGER WHEN DISTANCE=1 DELAY=-1 DO Schrittmerker_R1Place(10254,10253,FPlace_R1_L4_S1_VP5,XPlace_R1_L4_S1_VP5) PRIO=-1
;FOLD PTP Place_R1_L4_S1_VP5 CONT Vel=12 % PPlace_R1_L4_S1_VP5 Tool[2]:Lower Gripper Base[1]:Rack1;%{PE}%R8.3.21,%MKUKATPBASIS,%CMOVE,%VPTP,%P 1:PTP, 2:Place_R1_L4_S1_VP5, 3:C_DIS, 5:12, 7:PPlace_R1_L4_S1_VP5
$BWDSTART=FALSE
PDAT_ACT= PPPlace_R1_L4_S1_VP5
FDAT_ACT= FPlace_R1_L4_S1_VP5
BAS(#PTP_PARAMS,12)
PTP XPlace_R1_L4_S1_VP5 C_DIS
;ENDFOLD
TRIGGER WHEN DISTANCE=1 DELAY=-1 DO Schrittmerker_R1Place(10255,10254,FPlace_R1_L4_S1_VP6,XPlace_R1_L4_S1_VP6) PRIO=-1
;FOLD PTP Place_R1_L4_S1_VP6 CONT Vel=12 % PPlace_R1_L4_S1_VP6 Tool[2]:Lower Gripper Base[1]:Rack1;%{PE}%R8.3.21,%MKUKATPBASIS,%CMOVE,%VPTP,%P 1:PTP, 2:Place_R1_L4_S1_VP6, 3:C_DIS, 5:12, 7:PPlace_R1_L4_S1_VP6
$BWDSTART=FALSE
PDAT_ACT= PPPlace_R1_L4_S1_VP6
FDAT_ACT= FPlace_R1_L4_S1_VP6
BAS(#PTP_PARAMS,12)
PTP XPlace_R1_L4_S1_VP6 C_DIS
;ENDFOLD
TRIGGER WHEN DISTANCE=1 DELAY=-1 DO Schrittmerker_R1Place(10256,10255,FPlace_R1_L4_S1_VP7,XPlace_R1_L4_S1_VP7) PRIO=-1
;FOLD PTP Place_R1_L4_S1_VP7 CONT Vel=12 % PPlace_R1_L4_S1_VP7 Tool[2]:Lower Gripper Base[1]:Rack1;%{PE}%R8.3.21,%MKUKATPBASIS,%CMOVE,%VPTP,%P 1:PTP, 2:Place_R1_L4_S1_VP7, 3:C_DIS, 5:12, 7:PPlace_R1_L4_S1_VP7
$BWDSTART=FALSE
PDAT_ACT= PPPlace_R1_L4_S1_VP7
FDAT_ACT= FPlace_R1_L4_S1_VP7
BAS(#PTP_PARAMS,12)
PTP XPlace_R1_L4_S1_VP7 C_DIS
;ENDFOLD
TRIGGER WHEN DISTANCE=1 DELAY=-1 DO Schrittmerker_R1Place(10257,10256,FPlace_R1_L4_S1_VP8,XPlace_R1_L4_S1_VP8) PRIO=-1
;FOLD PTP Place_R1_L4_S1_VP8 CONT Vel=12 % PPlace_R1_L4_S1_VP8 Tool[2]:Lower Gripper Base[1]:Rack1;%{PE}%R8.3.21,%MKUKATPBASIS,%CMOVE,%VPTP,%P 1:PTP, 2:Place_R1_L4_S1_VP8, 3:C_DIS, 5:12, 7:PPlace_R1_L4_S1_VP8
$BWDSTART=FALSE
PDAT_ACT= PPPlace_R1_L4_S1_VP8
FDAT_ACT= FPlace_R1_L4_S1_VP8
BAS(#PTP_PARAMS,12)
PTP XPlace_R1_L4_S1_VP8 C_DIS
;ENDFOLD

TRIGGER WHEN DISTANCE=1 DELAY=-1 DO Schrittmerker_R1Place(10258,10257,FPlace_R1_L4_S1_Check,XPlace_R1_L4_S1_Check) PRIO=-1
;FOLD PTP Place_R1_L4_S1_Check Vel=12 % PPlace_R1_L4_S1_Check Tool[2]:Lower Gripper Base[1]:Rack1;%{PE}%R8.3.21,%MKUKATPBASIS,%CMOVE,%VPTP,%P 1:PTP, 2:Place_R1_L4_S1_Check, 3:, 5:12, 7:PPlace_R1_L4_S1_Check
$BWDSTART=FALSE
PDAT_ACT= PPPlace_R1_L4_S1_Check
FDAT_ACT= FPlace_R1_L4_S1_Check
BAS(#PTP_PARAMS,12)
PTP XPlace_R1_L4_S1_Check
;ENDFOLD

;***************************************************
;FOLD Pruefe Platz frei
IF (DetectPart(CHECK_SHELF,PLACE)==OCCUPIED) THEN
  UP_Rueckzug_R1Place( )
  RETURN
ENDIF
;ENDFOLD
;***************************************************

TRIGGER WHEN DISTANCE=1 DELAY=-1 DO Schrittmerker_R1Place(10259,10258,FPlace_R1_L4_S1_VP9,XPlace_R1_L4_S1_VP9) PRIO=-1
;FOLD LIN Place_R1_L4_S1_VP9 CONT Vel=0.5 m/s LPlace_R1_L4_S1_VP9 Tool[2]:Lower Gripper Base[1]:Rack1;%{PE}%R8.3.21,%MKUKATPBASIS,%CMOVE,%VLIN,%P 1:LIN, 2:Place_R1_L4_S1_VP9, 3:C_DIS C_DIS, 5:0.5, 7:LPlace_R1_L4_S1_VP9
$BWDSTART=FALSE
LDAT_ACT= LLPlace_R1_L4_S1_VP9
FDAT_ACT= FPlace_R1_L4_S1_VP9
BAS(#CP_PARAMS,0.5)
LIN XPlace_R1_L4_S1_VP9 C_DIS C_DIS
;ENDFOLD
TRIGGER WHEN DISTANCE=1 DELAY=-1 DO Schrittmerker_R1Place(10260,10259,FPlace_R1_L4_S1_VP10,XPlace_R1_L4_S1_VP10) PRIO=-1
;FOLD LIN Place_R1_L4_S1_VP10 CONT Vel=0.5 m/s LPlace_R1_L4_S1_VP10 Tool[2]:Lower Gripper Base[1]:Rack1;%{PE}%R8.3.21,%MKUKATPBASIS,%CMOVE,%VLIN,%P 1:LIN, 2:Place_R1_L4_S1_VP10, 3:C_DIS C_DIS, 5:0.5, 7:LPlace_R1_L4_S1_VP10
$BWDSTART=FALSE
LDAT_ACT= LLPlace_R1_L4_S1_VP10
FDAT_ACT= FPlace_R1_L4_S1_VP10
BAS(#CP_PARAMS,0.5)
LIN XPlace_R1_L4_S1_VP10 C_DIS C_DIS
;ENDFOLD

;FOLD Test the way back home - part 1
CONTINUE
IF ($FLAG[M_Test_GrdstFahren1] AND NOT $FLAG[M_Test_GrdstFahren2]) THEN
  $FLAG[M_Test_GrdstFahren2]=TRUE
  UP_Rueckzug( )
  RETURN
ENDIF
;ENDFOLD

;-------------------------------
; Place part position
;-------------------------------
TRIGGER WHEN DISTANCE=1 DELAY=-1 DO Schrittmerker_R1Place(10261,10262,FPlace_R1_L4_S1_AP,XPlace_R1_L4_S1_AP) PRIO=-1
;FOLD LIN Place_R1_L4_S1_AP Vel=0.2 m/s LPlace_R1_L4_S1_AP Tool[2]:Lower Gripper Base[1]:Rack1;%{PE}%R8.3.21,%MKUKATPBASIS,%CMOVE,%VLIN,%P 1:LIN, 2:Place_R1_L4_S1_AP, 3:, 5:0.2, 7:LPlace_R1_L4_S1_AP
$BWDSTART=FALSE
LDAT_ACT= LLPlace_R1_L4_S1_AP
FDAT_ACT= FPlace_R1_L4_S1_AP
BAS(#CP_PARAMS,0.2)
LIN XPlace_R1_L4_S1_AP
;ENDFOLD

;FOLD Test the way back home - part 2
CONTINUE
IF $FLAG[M_Test_GrdstFahren2] THEN
  $FLAG[M_Test_GrdstFahren2]=FALSE
  UP_Rueckzug( )
  RETURN
ENDIF
;ENDFOLD

;***************************************************
; Disable part lost detection
SetPartLostDetection(NO_PART)
;***************************************************

TRIGGER WHEN DISTANCE=1 DELAY=-1 DO Schrittmerker_R1Place(10262,10263,FPlace_R1_L4_S1_NP1,XPlace_R1_L4_S1_NP1) PRIO=-1
;FOLD LIN Place_R1_L4_S1_NP1 Vel=0.2 m/s LPlace_R1_L4_S1_NP1 Tool[2]:Lower Gripper Base[1]:Rack1;%{PE}%R8.3.21,%MKUKATPBASIS,%CMOVE,%VLIN,%P 1:LIN, 2:Place_R1_L4_S1_NP1, 3:C_DIS C_DIS, 5:0.2, 7:LPlace_R1_L4_S1_NP1
$BWDSTART=FALSE
LDAT_ACT= LLPlace_R1_L4_S1_NP1
FDAT_ACT= FPlace_R1_L4_S1_NP1
BAS(#CP_PARAMS,0.2)
LIN XPlace_R1_L4_S1_NP1
;ENDFOLD

;***************************************************
; Check for part present (empty gripper)
CheckPartPresent(EMPTY_GRIPPER)
;***************************************************
; set load data
SetLoadData( )
;***************************************************

TRIGGER WHEN DISTANCE=1 DELAY=-1 DO Schrittmerker_R1Place(10263,10264,FPlace_R1_L4_S1_NP2,XPlace_R1_L4_S1_NP2) PRIO=-1
;FOLD LIN Place_R1_L4_S1_NP2 CONT Vel=0.5 m/s LPlace_R1_L4_S1_NP2 Tool[2]:Lower Gripper Base[1]:Rack1;%{PE}%R8.3.21,%MKUKATPBASIS,%CMOVE,%VLIN,%P 1:LIN, 2:Place_R1_L4_S1_NP2, 3:C_DIS C_DIS, 5:0.5, 7:LPlace_R1_L4_S1_NP2
$BWDSTART=FALSE
LDAT_ACT= LLPlace_R1_L4_S1_NP2
FDAT_ACT= FPlace_R1_L4_S1_NP2
BAS(#CP_PARAMS,0.5)
LIN XPlace_R1_L4_S1_NP2 C_DIS C_DIS
;ENDFOLD
TRIGGER WHEN DISTANCE=1 DELAY=-1 DO Schrittmerker_R1Place(10264,10265,FPlace_R1_L4_S1_NP3,XPlace_R1_L4_S1_NP3) PRIO=-1
;FOLD LIN Place_R1_L4_S1_NP3 Vel=0.5 m/s LPlace_R1_L4_S1_NP3 Tool[2]:Lower Gripper Base[1]:Rack1;%{PE}%R8.3.21,%MKUKATPBASIS,%CMOVE,%VLIN,%P 1:LIN, 2:Place_R1_L4_S1_NP3, 3:, 5:0.5, 7:LPlace_R1_L4_S1_NP3
$BWDSTART=FALSE
LDAT_ACT= LLPlace_R1_L4_S1_NP3
FDAT_ACT= FPlace_R1_L4_S1_NP3
BAS(#CP_PARAMS,0.5)
LIN XPlace_R1_L4_S1_NP3
;ENDFOLD
TRIGGER WHEN DISTANCE=1 DELAY=-1 DO Schrittmerker_R1Place(10265,10266,FPlace_R1_L4_S1_NP4,XPlace_R1_L4_S1_NP4) PRIO=-1
;FOLD PTP Place_R1_L4_S1_NP4 CONT Vel=100 % PPlace_R1_L4_S1_NP4 Tool[2]:Lower Gripper Base[0];%{PE}%R8.3.21,%MKUKATPBASIS,%CMOVE,%VPTP,%P 1:PTP, 2:Place_R1_L4_S1_NP4, 3:C_DIS, 5:100, 7:PPlace_R1_L4_S1_NP4
$BWDSTART=FALSE
PDAT_ACT= PPPlace_R1_L4_S1_NP4
FDAT_ACT= FPlace_R1_L4_S1_NP4
BAS(#PTP_PARAMS,100)
PTP XPlace_R1_L4_S1_NP4 C_DIS
;ENDFOLD
TRIGGER WHEN DISTANCE=1 DELAY=-1 DO Schrittmerker_R1Place(10266,10267,FPlace_R1_L4_S1_NP5,XPlace_R1_L4_S1_NP5) PRIO=-1
;FOLD PTP Place_R1_L4_S1_NP5 CONT Vel=100 % PPlace_R1_L4_S1_NP5 Tool[2]:Lower Gripper Base[0];%{PE}%R8.3.21,%MKUKATPBASIS,%CMOVE,%VPTP,%P 1:PTP, 2:Place_R1_L4_S1_NP5, 3:C_DIS, 5:100, 7:PPlace_R1_L4_S1_NP5
$BWDSTART=FALSE
PDAT_ACT= PPPlace_R1_L4_S1_NP5
FDAT_ACT= FPlace_R1_L4_S1_NP5
BAS(#PTP_PARAMS,100)
PTP XPlace_R1_L4_S1_NP5 C_DIS
;ENDFOLD
TRIGGER WHEN DISTANCE=1 DELAY=-1 DO Schrittmerker_R1Place(10267,10268,FPlace_R1_L4_S1_NP6,XPlace_R1_L4_S1_NP6) PRIO=-1
;FOLD PTP Place_R1_L4_S1_NP6 CONT Vel=100 % PPlace_R1_L4_S1_NP6 Tool[2]:Lower Gripper Base[0];%{PE}
;FOLD Parameters ;%{h}
;Params IlfProvider=kukaroboter.basistech.inlineforms.movement.old; Kuka.IsGlobalPoint=False; Kuka.PointName=Place_R1_L4_S1_NP6; Kuka.BlendingEnabled=True; Kuka.MoveDataPtpName=PPlace_R1_L4_S1_NP6; Kuka.VelocityPtp=100; Kuka.CurrentCDSetIndex=0; Kuka.MovementParameterFieldEnabled=True; IlfCommand=PTP
;ENDFOLD
$BWDSTART = FALSE
PDAT_ACT = PPPlace_R1_L4_S1_NP6
FDAT_ACT = FPlace_R1_L4_S1_NP6
BAS(#PTP_PARAMS, 100.0)
SET_CD_PARAMS (0)
PTP XPlace_R1_L4_S1_NP6 C_Dis
;ENDFOLD

TRIGGER WHEN DISTANCE=1 DELAY=-1 DO Schrittmerker_R1Place(10268,10002,FHOME1,$nullframe,XHOME1) PRIO=-1
;FOLD PTP HOME1 Vel=100 % PHome1;%{PE}%R8.3.21,%MKUKATPBASIS,%CMOVE,%VPTP,%P 1:PTP, 2:HOME1, 3:, 5:100, 7:PHome1
$BWDSTART=FALSE
PDAT_ACT= PPHome1
FDAT_ACT= FHOME1
BAS(#PTP_PARAMS,100)
PTP XHOME1
;ENDFOLD

;***************************************************
;FOLD Final tasks.
; Robot out of area Rack 1 Level 4
RobAusStorage1_4_A70=RESET_IN_AREA
;***************************************************
; stop cyclic clearence check
$CYCFLAG[ciFreigabeSPS]=DISABLE_MONITORING
;***************************************************
; Disable collision detection
;FOLD COLLDETECT Off ;%{PE}
;FOLD Parameters ;%{h}
;Params IlfProvider=kukaroboter.basistech.inlineforms.colldetect.off; CollDetect.Command=Off
;ENDFOLD
USE_CD_PARAMS(0)
;ENDFOLD
;***************************************************
;ENDFOLD
;***************************************************

END

; ##################################################

GLOBAL DEF UP_Place_R1_L4_S2( )
;***************************************************
; Place part on:
;    Rack  1
;    Level 4
;    Shelf 2
;***************************************************
;FOLD Preconditions - Vorraussetzungen
;***************************************************
; Enable collision detection
;FOLD COLLDETECT SetLimits Axis1: 150 % Axis2: 200 % Axis3: 150 % Axis4: 200 % Axis5: 150 % Axis6: 150 % ;%{PE}
;FOLD Parameters ;%{h}
;Params IlfProvider=kukaroboter.basistech.inlineforms.colldetect.setlimits; CollDetect.Command=SetLimits; CollDetect.Axis1=150; CollDetect.Axis2=200; CollDetect.Axis3=150; CollDetect.Axis4=200; CollDetect.Axis5=150; CollDetect.Axis6=150
;ENDFOLD
SET_TQ_VALUES(150, 200, 150, 200, 150, 150)
;ENDFOLD
;***************************************************
; Check for part in gripper (tool 2).
CheckPartPresent(OCCUPIED_GRIPPER,PART_ON_TOOL_2)
;***************************************************
; Enable part lost detection for tool 2
SetPartLostDetection(PART_ON_TOOL_2)
;***************************************************
; Set load data.
SetLoadData( )
;***************************************************
; Robot has to start from home position.
IF NOT $IN_HOME1 THEN
  UP_HomeToHome(1)
ENDIF
;***************************************************
;ENDFOLD

TRIGGER WHEN DISTANCE=1 DELAY=-1 DO Schrittmerker_R1Place(10002,10002,FHOME1,$nullframe,XHOME1) PRIO=-1
;FOLD PTP HOME1 Vel=12 % PHome1;%{PE}%R8.3.21,%MKUKATPBASIS,%CMOVE,%VPTP,%P 1:PTP, 2:HOME1, 3:, 5:12, 7:PHome1
$BWDSTART=FALSE
PDAT_ACT= PPHome1
FDAT_ACT= FHOME1
BAS(#PTP_PARAMS,12)
PTP XHOME1
;ENDFOLD

;***************************************************
;FOLD Area clearence handshake.
IF NOT $FLAG[M_Inbetriebnahme] THEN
  ;-------------------------------------------------
  ; Request area clearence.
  AnfStoer_Store1_4_A102=SET_REQUEST
  ;-------------------------------------------------
  ; Wait for area clearence from PLC.
  WAIT_FOR_INPUT("Frg_Storage1_4_E70",TRUE)
  ;-------------------------------------------------
  ; Reset area clearence request.
  AnfStoer_Store1_4_A102=RESET_REQUEST
  ;-------------------------------------------------
  ; start cyclic clearence check
  $CYCFLAG[ciFreigabeSPS]=Frg_Storage1_4_E70
  ;-------------------------------------------------
ENDIF
;***************************************************
; set "robot in area"
RobAusStorage1_4_A70=SET_IN_AREA
;ENDFOLD
;***************************************************

;***************************************************
;FOLD Check for Teachmode
IF $FLAG[M_Teachen] THEN
  WAIT FOR $T1
ENDIF
;ENDFOLD
;***************************************************

; move to the rack
TRIGGER WHEN DISTANCE=1 DELAY=-1 DO Schrittmerker_R1Place(10270,10002,FPlace_R1_L4_S2_VP1,XPlace_R1_L4_S2_VP1) PRIO=-1
;FOLD PTP Place_R1_L4_S2_VP1 CONT Vel=12 % PPlace_R1_L4_S2_VP1 Tool[2]:Lower Gripper Base[0];%{PE}%R8.3.21,%MKUKATPBASIS,%CMOVE,%VPTP,%P 1:PTP, 2:Place_R1_L4_S2_VP1, 3:C_DIS, 5:12, 7:PPlace_R1_L4_S2_VP1
$BWDSTART=FALSE
PDAT_ACT= PPPlace_R1_L4_S2_VP1
FDAT_ACT= FPlace_R1_L4_S2_VP1
BAS(#PTP_PARAMS,12)
PTP XPlace_R1_L4_S2_VP1 C_DIS
;ENDFOLD
TRIGGER WHEN DISTANCE=1 DELAY=-1 DO Schrittmerker_R1Place(10271,10270,FPlace_R1_L4_S2_VP2,XPlace_R1_L4_S2_VP2) PRIO=-1
;FOLD PTP Place_R1_L4_S2_VP2 CONT Vel=12 % PPlace_R1_L4_S2_VP2 Tool[2]:Lower Gripper Base[0];%{PE}%R8.3.21,%MKUKATPBASIS,%CMOVE,%VPTP,%P 1:PTP, 2:Place_R1_L4_S2_VP2, 3:C_DIS, 5:12, 7:PPlace_R1_L4_S2_VP2
$BWDSTART=FALSE
PDAT_ACT= PPPlace_R1_L4_S2_VP2
FDAT_ACT= FPlace_R1_L4_S2_VP2
BAS(#PTP_PARAMS,12)
PTP XPlace_R1_L4_S2_VP2 C_DIS
;ENDFOLD
TRIGGER WHEN DISTANCE=1 DELAY=-1 DO Schrittmerker_R1Place(10272,10271,FPlace_R1_L4_S2_VP3,XPlace_R1_L4_S2_VP3) PRIO=-1
;FOLD PTP Place_R1_L4_S2_VP3 CONT Vel=12 % PPlace_R1_L4_S2_VP3 Tool[2]:Lower Gripper Base[0];%{PE}%R8.3.21,%MKUKATPBASIS,%CMOVE,%VPTP,%P 1:PTP, 2:Place_R1_L4_S2_VP3, 3:C_DIS, 5:12, 7:PPlace_R1_L4_S2_VP3
$BWDSTART=FALSE
PDAT_ACT= PPPlace_R1_L4_S2_VP3
FDAT_ACT= FPlace_R1_L4_S2_VP3
BAS(#PTP_PARAMS,12)
PTP XPlace_R1_L4_S2_VP3 C_DIS
;ENDFOLD
TRIGGER WHEN DISTANCE=1 DELAY=-1 DO Schrittmerker_R1Place(10273,10272,FPlace_R1_L4_S2_VP4,XPlace_R1_L4_S2_VP4) PRIO=-1
;FOLD PTP Place_R1_L4_S2_VP4 CONT Vel=12 % PPlace_R1_L4_S2_VP4 Tool[2]:Lower Gripper Base[1]:Rack1;%{PE}%R8.3.21,%MKUKATPBASIS,%CMOVE,%VPTP,%P 1:PTP, 2:Place_R1_L4_S2_VP4, 3:C_DIS, 5:12, 7:PPlace_R1_L4_S2_VP4
$BWDSTART=FALSE
PDAT_ACT= PPPlace_R1_L4_S2_VP4
FDAT_ACT= FPlace_R1_L4_S2_VP4
BAS(#PTP_PARAMS,12)
PTP XPlace_R1_L4_S2_VP4 C_DIS
;ENDFOLD

TRIGGER WHEN DISTANCE=1 DELAY=-1 DO Schrittmerker_R1Place(10274,10273,FPlace_R1_L4_S2_Check,XPlace_R1_L4_S2_Check) PRIO=-1
;FOLD PTP Place_R1_L4_S2_Check Vel=12 % PPlace_R1_L4_S2_Check Tool[2]:Lower Gripper Base[1]:Rack1;%{PE}%R8.3.21,%MKUKATPBASIS,%CMOVE,%VPTP,%P 1:PTP, 2:Place_R1_L4_S2_Check, 3:, 5:12, 7:PPlace_R1_L4_S2_Check
$BWDSTART=FALSE
PDAT_ACT= PPPlace_R1_L4_S2_Check
FDAT_ACT= FPlace_R1_L4_S2_Check
BAS(#PTP_PARAMS,12)
PTP XPlace_R1_L4_S2_Check
;ENDFOLD

;***************************************************
;FOLD Pruefe Platz frei
IF (DetectPart(CHECK_SHELF,PLACE)==OCCUPIED) THEN
  UP_Rueckzug_R1Place( )
  RETURN
ENDIF
;ENDFOLD
;***************************************************

TRIGGER WHEN DISTANCE=1 DELAY=-1 DO Schrittmerker_R1Place(10275,10274,FPlace_R1_L4_S2_VP5,XPlace_R1_L4_S2_VP5) PRIO=-1
;FOLD LIN Place_R1_L4_S2_VP5 CONT Vel=0.5 m/s LPlace_R1_L4_S2_VP5 Tool[2]:Lower Gripper Base[1]:Rack1;%{PE}%R8.3.21,%MKUKATPBASIS,%CMOVE,%VLIN,%P 1:LIN, 2:Place_R1_L4_S2_VP5, 3:C_DIS C_DIS, 5:0.5, 7:LPlace_R1_L4_S2_VP5
$BWDSTART=FALSE
LDAT_ACT= LLPlace_R1_L4_S2_VP5
FDAT_ACT= FPlace_R1_L4_S2_VP5
BAS(#CP_PARAMS,0.5)
LIN XPlace_R1_L4_S2_VP5 C_DIS C_DIS
;ENDFOLD
TRIGGER WHEN DISTANCE=1 DELAY=-1 DO Schrittmerker_R1Place(10276,10275,FPlace_R1_L4_S2_VP6,XPlace_R1_L4_S2_VP6) PRIO=-1
;FOLD LIN Place_R1_L4_S2_VP6 CONT Vel=0.5 m/s LPlace_R1_L4_S2_VP6 Tool[2]:Lower Gripper Base[1]:Rack1;%{PE}%R8.3.21,%MKUKATPBASIS,%CMOVE,%VLIN,%P 1:LIN, 2:Place_R1_L4_S2_VP6, 3:C_DIS C_DIS, 5:0.5, 7:LPlace_R1_L4_S2_VP6
$BWDSTART=FALSE
LDAT_ACT= LLPlace_R1_L4_S2_VP6
FDAT_ACT= FPlace_R1_L4_S2_VP6
BAS(#CP_PARAMS,0.5)
LIN XPlace_R1_L4_S2_VP6 C_DIS C_DIS
;ENDFOLD
TRIGGER WHEN DISTANCE=1 DELAY=-1 DO Schrittmerker_R1Place(10277,10276,FPlace_R1_L4_S2_VP7,XPlace_R1_L4_S2_VP7) PRIO=-1
;FOLD LIN Place_R1_L4_S2_VP7 CONT Vel=0.5 m/s LPlace_R1_L4_S2_VP7 Tool[2]:Lower Gripper Base[1]:Rack1;%{PE}%R8.3.21,%MKUKATPBASIS,%CMOVE,%VLIN,%P 1:LIN, 2:Place_R1_L4_S2_VP7, 3:C_DIS C_DIS, 5:0.5, 7:LPlace_R1_L4_S2_VP7
$BWDSTART=FALSE
LDAT_ACT= LLPlace_R1_L4_S2_VP7
FDAT_ACT= FPlace_R1_L4_S2_VP7
BAS(#CP_PARAMS,0.5)
LIN XPlace_R1_L4_S2_VP7 C_DIS C_DIS
;ENDFOLD

;FOLD Test the way back home - part 1
CONTINUE
IF ($FLAG[M_Test_GrdstFahren1] AND NOT $FLAG[M_Test_GrdstFahren2]) THEN
  $FLAG[M_Test_GrdstFahren2]=TRUE
  UP_Rueckzug( )
  RETURN
ENDIF
;ENDFOLD

;-------------------------------
; Place part position
;-------------------------------
TRIGGER WHEN DISTANCE=1 DELAY=-1 DO Schrittmerker_R1Place(10278,10279,FPlace_R1_L4_S2_AP,XPlace_R1_L4_S2_AP) PRIO=-1
;FOLD LIN Place_R1_L4_S2_AP Vel=0.2 m/s LPlace_R1_L4_S2_AP Tool[2]:Lower Gripper Base[1]:Rack1;%{PE}%R8.3.21,%MKUKATPBASIS,%CMOVE,%VLIN,%P 1:LIN, 2:Place_R1_L4_S2_AP, 3:, 5:0.2, 7:LPlace_R1_L4_S2_AP
$BWDSTART=FALSE
LDAT_ACT= LLPlace_R1_L4_S2_AP
FDAT_ACT= FPlace_R1_L4_S2_AP
BAS(#CP_PARAMS,0.2)
LIN XPlace_R1_L4_S2_AP
;ENDFOLD

;FOLD Test the way back home - part 2
CONTINUE
IF $FLAG[M_Test_GrdstFahren2] THEN
  $FLAG[M_Test_GrdstFahren2]=FALSE
  UP_Rueckzug( )
  RETURN
ENDIF
;ENDFOLD

;***************************************************
; Disable part lost detection
SetPartLostDetection(NO_PART)
;***************************************************

TRIGGER WHEN DISTANCE=1 DELAY=-1 DO Schrittmerker_R1Place(10279,10280,FPlace_R1_L4_S2_NP1,XPlace_R1_L4_S2_NP1) PRIO=-1
;FOLD LIN Place_R1_L4_S2_NP1 Vel=0.2 m/s LPlace_R1_L4_S2_NP1 Tool[2]:Lower Gripper Base[1]:Rack1;%{PE}%R8.3.21,%MKUKATPBASIS,%CMOVE,%VLIN,%P 1:LIN, 2:Place_R1_L4_S2_NP1, 3:C_DIS C_DIS, 5:0.2, 7:LPlace_R1_L4_S2_NP1
$BWDSTART=FALSE
LDAT_ACT= LLPlace_R1_L4_S2_NP1
FDAT_ACT= FPlace_R1_L4_S2_NP1
BAS(#CP_PARAMS,0.2)
LIN XPlace_R1_L4_S2_NP1
;ENDFOLD

;***************************************************
; Check for part present (empty gripper)
CheckPartPresent(EMPTY_GRIPPER)
;***************************************************
; set load data
SetLoadData( )
;***************************************************

TRIGGER WHEN DISTANCE=1 DELAY=-1 DO Schrittmerker_R1Place(10280,10281,FPlace_R1_L4_S2_NP2,XPlace_R1_L4_S2_NP2) PRIO=-1
;FOLD LIN Place_R1_L4_S2_NP2 Vel=0.5 m/s LPlace_R1_L4_S2_NP2 Tool[2]:Lower Gripper Base[1]:Rack1;%{PE}%R8.3.21,%MKUKATPBASIS,%CMOVE,%VLIN,%P 1:LIN, 2:Place_R1_L4_S2_NP2, 3:, 5:0.5, 7:LPlace_R1_L4_S2_NP2
$BWDSTART=FALSE
LDAT_ACT= LLPlace_R1_L4_S2_NP2
FDAT_ACT= FPlace_R1_L4_S2_NP2
BAS(#CP_PARAMS,0.5)
LIN XPlace_R1_L4_S2_NP2
;ENDFOLD
TRIGGER WHEN DISTANCE=1 DELAY=-1 DO Schrittmerker_R1Place(10281,10282,FPlace_R1_L4_S2_NP3,XPlace_R1_L4_S2_NP3) PRIO=-1
;FOLD PTP Place_R1_L4_S2_NP3 CONT Vel=100 % PPlace_R1_L4_S2_NP3 Tool[2]:Lower Gripper Base[0];%{PE}%R8.3.21,%MKUKATPBASIS,%CMOVE,%VPTP,%P 1:PTP, 2:Place_R1_L4_S2_NP3, 3:C_DIS, 5:100, 7:PPlace_R1_L4_S2_NP3
$BWDSTART=FALSE
PDAT_ACT= PPPlace_R1_L4_S2_NP3
FDAT_ACT= FPlace_R1_L4_S2_NP3
BAS(#PTP_PARAMS,100)
PTP XPlace_R1_L4_S2_NP3 C_DIS
;ENDFOLD
TRIGGER WHEN DISTANCE=1 DELAY=-1 DO Schrittmerker_R1Place(10282,10283,FPlace_R1_L4_S2_NP4,XPlace_R1_L4_S2_NP4) PRIO=-1
;FOLD PTP Place_R1_L4_S2_NP4 CONT Vel=100 % PPlace_R1_L4_S2_NP4 Tool[2]:Lower Gripper Base[0];%{PE}%R8.3.21,%MKUKATPBASIS,%CMOVE,%VPTP,%P 1:PTP, 2:Place_R1_L4_S2_NP4, 3:C_DIS, 5:100, 7:PPlace_R1_L4_S2_NP4
$BWDSTART=FALSE
PDAT_ACT= PPPlace_R1_L4_S2_NP4
FDAT_ACT= FPlace_R1_L4_S2_NP4
BAS(#PTP_PARAMS,100)
PTP XPlace_R1_L4_S2_NP4 C_DIS
;ENDFOLD
TRIGGER WHEN DISTANCE=1 DELAY=-1 DO Schrittmerker_R1Place(10283,10284,FPlace_R1_L4_S2_NP5,XPlace_R1_L4_S2_NP5) PRIO=-1
;FOLD PTP Place_R1_L4_S2_NP5 CONT Vel=100 % PPlace_R1_L4_S2_NP5 Tool[2]:Lower Gripper Base[0];%{PE}%R8.3.21,%MKUKATPBASIS,%CMOVE,%VPTP,%P 1:PTP, 2:Place_R1_L4_S2_NP5, 3:C_DIS, 5:100, 7:PPlace_R1_L4_S2_NP5
$BWDSTART=FALSE
PDAT_ACT= PPPlace_R1_L4_S2_NP5
FDAT_ACT= FPlace_R1_L4_S2_NP5
BAS(#PTP_PARAMS,100)
PTP XPlace_R1_L4_S2_NP5 C_DIS
;ENDFOLD
TRIGGER WHEN DISTANCE=1 DELAY=-1 DO Schrittmerker_R1Place(10284,10285,FPlace_R1_L4_S2_NP6,XPlace_R1_L4_S2_NP6) PRIO=-1
;FOLD PTP Place_R1_L4_S2_NP6 CONT Vel=100 % PPlace_R1_L4_S2_NP6 Tool[2]:Lower Gripper Base[0];%{PE}
;FOLD Parameters ;%{h}
;Params IlfProvider=kukaroboter.basistech.inlineforms.movement.old; Kuka.IsGlobalPoint=False; Kuka.PointName=Place_R1_L4_S2_NP6; Kuka.BlendingEnabled=True; Kuka.MoveDataPtpName=PPlace_R1_L4_S2_NP6; Kuka.VelocityPtp=100; Kuka.CurrentCDSetIndex=0; Kuka.MovementParameterFieldEnabled=True; IlfCommand=PTP
;ENDFOLD
$BWDSTART = FALSE
PDAT_ACT = PPPlace_R1_L4_S2_NP6
FDAT_ACT = FPlace_R1_L4_S2_NP6
BAS(#PTP_PARAMS, 100.0)
SET_CD_PARAMS (0)
PTP XPlace_R1_L4_S2_NP6 C_Dis
;ENDFOLD

TRIGGER WHEN DISTANCE=1 DELAY=-1 DO Schrittmerker_R1Place(10285,10002,FHOME1,$nullframe,XHOME1) PRIO=-1
;FOLD PTP HOME1 Vel=100 % PHome1;%{PE}%R8.3.21,%MKUKATPBASIS,%CMOVE,%VPTP,%P 1:PTP, 2:HOME1, 3:, 5:100, 7:PHome1
$BWDSTART=FALSE
PDAT_ACT= PPHome1
FDAT_ACT= FHOME1
BAS(#PTP_PARAMS,100)
PTP XHOME1
;ENDFOLD

;***************************************************
;FOLD Final tasks.
; Robot out of area Rack 1 Level 4
RobAusStorage1_4_A70=RESET_IN_AREA
;***************************************************
; stop cyclic clearence check
$CYCFLAG[ciFreigabeSPS]=DISABLE_MONITORING
;***************************************************
; Disable collision detection
;FOLD COLLDETECT Off ;%{PE}
;FOLD Parameters ;%{h}
;Params IlfProvider=kukaroboter.basistech.inlineforms.colldetect.off; CollDetect.Command=Off
;ENDFOLD
USE_CD_PARAMS(0)
;ENDFOLD
;***************************************************
;ENDFOLD
;***************************************************

END

; ##################################################

GLOBAL DEF UP_Place_R1_L4_S3( )
;***************************************************
; Place part on:
;    Rack  1
;    Level 4
;    Shelf 3
;***************************************************
;FOLD Preconditions - Vorraussetzungen
;***************************************************
; Enable collision detection
;FOLD COLLDETECT SetLimits Axis1: 150 % Axis2: 200 % Axis3: 150 % Axis4: 200 % Axis5: 150 % Axis6: 150 % ;%{PE}
;FOLD Parameters ;%{h}
;Params IlfProvider=kukaroboter.basistech.inlineforms.colldetect.setlimits; CollDetect.Command=SetLimits; CollDetect.Axis1=150; CollDetect.Axis2=200; CollDetect.Axis3=150; CollDetect.Axis4=200; CollDetect.Axis5=150; CollDetect.Axis6=150
;ENDFOLD
SET_TQ_VALUES(150, 200, 150, 200, 150, 150)
;ENDFOLD
;***************************************************
; Check for part in gripper (tool 2).
CheckPartPresent(OCCUPIED_GRIPPER,PART_ON_TOOL_2)
;***************************************************
; Enable part lost detection for tool 2
SetPartLostDetection(PART_ON_TOOL_2)
;***************************************************
; Set load data.
SetLoadData( )
;***************************************************
; Robot has to start from home position.
IF NOT $IN_HOME1 THEN
  UP_HomeToHome(1)
ENDIF
;***************************************************
;ENDFOLD

TRIGGER WHEN DISTANCE=1 DELAY=-1 DO Schrittmerker_R1Place(10002,10002,FHOME1,$nullframe,XHOME1) PRIO=-1
;FOLD PTP HOME1 Vel=12 % PHome1;%{PE}%R8.3.21,%MKUKATPBASIS,%CMOVE,%VPTP,%P 1:PTP, 2:HOME1, 3:, 5:12, 7:PHome1
$BWDSTART=FALSE
PDAT_ACT= PPHome1
FDAT_ACT= FHOME1
BAS(#PTP_PARAMS,12)
PTP XHOME1
;ENDFOLD

;***************************************************
;FOLD Area clearence handshake.
IF NOT $FLAG[M_Inbetriebnahme] THEN
  ;-------------------------------------------------
  ; Request area clearence.
  AnfStoer_Store1_4_A102=SET_REQUEST
  ;-------------------------------------------------
  ; Wait for area clearence from PLC.
  WAIT_FOR_INPUT("Frg_Storage1_4_E70",TRUE)
  ;-------------------------------------------------
  ; Reset area clearence request.
  AnfStoer_Store1_4_A102=RESET_REQUEST
  ;-------------------------------------------------
  ; start cyclic clearence check
  $CYCFLAG[ciFreigabeSPS]=Frg_Storage1_4_E70
  ;-------------------------------------------------
ENDIF
;***************************************************
; set "robot in area"
RobAusStorage1_4_A70=SET_IN_AREA
;ENDFOLD
;***************************************************

;***************************************************
;FOLD Check for Teachmode
IF $FLAG[M_Teachen] THEN
  WAIT FOR $T1
ENDIF
;ENDFOLD
;***************************************************

; move to the rack
TRIGGER WHEN DISTANCE=1 DELAY=-1 DO Schrittmerker_R1Place(10290,10002,FPlace_R1_L4_S3_VP1,XPlace_R1_L4_S3_VP1) PRIO=-1
;FOLD PTP Place_R1_L4_S3_VP1 CONT Vel=12 % PPlace_R1_L4_S3_VP1 Tool[2]:Lower Gripper Base[0];%{PE}%R8.3.21,%MKUKATPBASIS,%CMOVE,%VPTP,%P 1:PTP, 2:Place_R1_L4_S3_VP1, 3:C_DIS, 5:12, 7:PPlace_R1_L4_S3_VP1
$BWDSTART=FALSE
PDAT_ACT= PPPlace_R1_L4_S3_VP1
FDAT_ACT= FPlace_R1_L4_S3_VP1
BAS(#PTP_PARAMS,12)
PTP XPlace_R1_L4_S3_VP1 C_DIS
;ENDFOLD
TRIGGER WHEN DISTANCE=1 DELAY=-1 DO Schrittmerker_R1Place(10291,10290,FPlace_R1_L4_S3_VP2,XPlace_R1_L4_S3_VP2) PRIO=-1
;FOLD PTP Place_R1_L4_S3_VP2 CONT Vel=12 % PPlace_R1_L4_S3_VP2 Tool[2]:Lower Gripper Base[0];%{PE}%R8.3.21,%MKUKATPBASIS,%CMOVE,%VPTP,%P 1:PTP, 2:Place_R1_L4_S3_VP2, 3:C_DIS, 5:12, 7:PPlace_R1_L4_S3_VP2
$BWDSTART=FALSE
PDAT_ACT= PPPlace_R1_L4_S3_VP2
FDAT_ACT= FPlace_R1_L4_S3_VP2
BAS(#PTP_PARAMS,12)
PTP XPlace_R1_L4_S3_VP2 C_DIS
;ENDFOLD
TRIGGER WHEN DISTANCE=1 DELAY=-1 DO Schrittmerker_R1Place(10292,10291,FPlace_R1_L4_S3_VP3,XPlace_R1_L4_S3_VP3) PRIO=-1
;FOLD PTP Place_R1_L4_S3_VP3 CONT Vel=12 % PPlace_R1_L4_S3_VP3 Tool[2]:Lower Gripper Base[0];%{PE}%R8.3.21,%MKUKATPBASIS,%CMOVE,%VPTP,%P 1:PTP, 2:Place_R1_L4_S3_VP3, 3:C_DIS, 5:12, 7:PPlace_R1_L4_S3_VP3
$BWDSTART=FALSE
PDAT_ACT= PPPlace_R1_L4_S3_VP3
FDAT_ACT= FPlace_R1_L4_S3_VP3
BAS(#PTP_PARAMS,12)
PTP XPlace_R1_L4_S3_VP3 C_DIS
;ENDFOLD

TRIGGER WHEN DISTANCE=1 DELAY=-1 DO Schrittmerker_R1Place(10293,10292,FPlace_R1_L4_S3_Check,XPlace_R1_L4_S3_Check) PRIO=-1
;FOLD PTP Place_R1_L4_S3_Check Vel=12 % PPlace_R1_L4_S3_Check Tool[2]:Lower Gripper Base[1]:Rack1;%{PE}%R8.3.21,%MKUKATPBASIS,%CMOVE,%VPTP,%P 1:PTP, 2:Place_R1_L4_S3_Check, 3:, 5:12, 7:PPlace_R1_L4_S3_Check
$BWDSTART=FALSE
PDAT_ACT= PPPlace_R1_L4_S3_Check
FDAT_ACT= FPlace_R1_L4_S3_Check
BAS(#PTP_PARAMS,12)
PTP XPlace_R1_L4_S3_Check
;ENDFOLD

;***************************************************
;FOLD Pruefe Platz frei
IF (DetectPart(CHECK_SHELF,PLACE)==OCCUPIED) THEN
  UP_Rueckzug_R1Place( )
  RETURN
ENDIF
;ENDFOLD
;***************************************************

TRIGGER WHEN DISTANCE=1 DELAY=-1 DO Schrittmerker_R1Place(10294,10293,FPlace_R1_L4_S3_VP4,XPlace_R1_L4_S3_VP4) PRIO=-1
;FOLD LIN Place_R1_L4_S3_VP4 CONT Vel=0.5 m/s LPlace_R1_L4_S3_VP4 Tool[2]:Lower Gripper Base[1]:Rack1;%{PE}%R8.3.21,%MKUKATPBASIS,%CMOVE,%VLIN,%P 1:LIN, 2:Place_R1_L4_S3_VP4, 3:C_DIS C_DIS, 5:0.5, 7:LPlace_R1_L4_S3_VP4
$BWDSTART=FALSE
LDAT_ACT= LLPlace_R1_L4_S3_VP4
FDAT_ACT= FPlace_R1_L4_S3_VP4
BAS(#CP_PARAMS,0.5)
LIN XPlace_R1_L4_S3_VP4 C_DIS C_DIS
;ENDFOLD
TRIGGER WHEN DISTANCE=1 DELAY=-1 DO Schrittmerker_R1Place(10295,10294,FPlace_R1_L4_S3_VP5,XPlace_R1_L4_S3_VP5) PRIO=-1
;FOLD LIN Place_R1_L4_S3_VP5 CONT Vel=0.5 m/s LPlace_R1_L4_S3_VP5 Tool[2]:Lower Gripper Base[1]:Rack1;%{PE}%R8.3.21,%MKUKATPBASIS,%CMOVE,%VLIN,%P 1:LIN, 2:Place_R1_L4_S3_VP5, 3:C_DIS C_DIS, 5:0.5, 7:LPlace_R1_L4_S3_VP5
$BWDSTART=FALSE
LDAT_ACT= LLPlace_R1_L4_S3_VP5
FDAT_ACT= FPlace_R1_L4_S3_VP5
BAS(#CP_PARAMS,0.5)
LIN XPlace_R1_L4_S3_VP5 C_DIS C_DIS
;ENDFOLD
TRIGGER WHEN DISTANCE=1 DELAY=-1 DO Schrittmerker_R1Place(10296,10295,FPlace_R1_L4_S3_VP6,XPlace_R1_L4_S3_VP6) PRIO=-1
;FOLD LIN Place_R1_L4_S3_VP6 CONT Vel=0.5 m/s LPlace_R1_L4_S3_VP6 Tool[2]:Lower Gripper Base[1]:Rack1;%{PE}%R8.3.21,%MKUKATPBASIS,%CMOVE,%VLIN,%P 1:LIN, 2:Place_R1_L4_S3_VP6, 3:C_DIS C_DIS, 5:0.5, 7:LPlace_R1_L4_S3_VP6
$BWDSTART=FALSE
LDAT_ACT= LLPlace_R1_L4_S3_VP6
FDAT_ACT= FPlace_R1_L4_S3_VP6
BAS(#CP_PARAMS,0.5)
LIN XPlace_R1_L4_S3_VP6 C_DIS C_DIS
;ENDFOLD

;FOLD Test the way back home - part 1
CONTINUE
IF ($FLAG[M_Test_GrdstFahren1] AND NOT $FLAG[M_Test_GrdstFahren2]) THEN
  $FLAG[M_Test_GrdstFahren2]=TRUE
  UP_Rueckzug( )
  RETURN
ENDIF
;ENDFOLD

;-------------------------------
; Place part position
;-------------------------------
TRIGGER WHEN DISTANCE=1 DELAY=-1 DO Schrittmerker_R1Place(10297,10298,FPlace_R1_L4_S3_AP,XPlace_R1_L4_S3_AP) PRIO=-1
;FOLD LIN Place_R1_L4_S3_AP Vel=0.2 m/s LPlace_R1_L4_S3_AP Tool[2]:Lower Gripper Base[1]:Rack1;%{PE}%R8.3.21,%MKUKATPBASIS,%CMOVE,%VLIN,%P 1:LIN, 2:Place_R1_L4_S3_AP, 3:, 5:0.2, 7:LPlace_R1_L4_S3_AP
$BWDSTART=FALSE
LDAT_ACT= LLPlace_R1_L4_S3_AP
FDAT_ACT= FPlace_R1_L4_S3_AP
BAS(#CP_PARAMS,0.2)
LIN XPlace_R1_L4_S3_AP
;ENDFOLD

;FOLD Test the way back home - part 2
CONTINUE
IF $FLAG[M_Test_GrdstFahren2] THEN
  $FLAG[M_Test_GrdstFahren2]=FALSE
  UP_Rueckzug( )
  RETURN
ENDIF
;ENDFOLD

;***************************************************
; Disable part lost detection
SetPartLostDetection(NO_PART)
;***************************************************

TRIGGER WHEN DISTANCE=1 DELAY=-1 DO Schrittmerker_R1Place(10298,10299,FPlace_R1_L4_S3_NP1,XPlace_R1_L4_S3_NP1) PRIO=-1
;FOLD LIN Place_R1_L4_S3_NP1 Vel=0.2 m/s LPlace_R1_L4_S3_NP1 Tool[2]:Lower Gripper Base[1]:Rack1;%{PE}%R8.3.21,%MKUKATPBASIS,%CMOVE,%VLIN,%P 1:LIN, 2:Place_R1_L4_S3_NP1, 3:C_DIS C_DIS, 5:0.2, 7:LPlace_R1_L4_S3_NP1
$BWDSTART=FALSE
LDAT_ACT= LLPlace_R1_L4_S3_NP1
FDAT_ACT= FPlace_R1_L4_S3_NP1
BAS(#CP_PARAMS,0.2)
LIN XPlace_R1_L4_S3_NP1
;ENDFOLD

;***************************************************
; Check for part present (empty gripper)
CheckPartPresent(EMPTY_GRIPPER)
;***************************************************
; set load data
SetLoadData( )
;***************************************************

TRIGGER WHEN DISTANCE=1 DELAY=-1 DO Schrittmerker_R1Place(10299,10300,FPlace_R1_L4_S3_NP2,XPlace_R1_L4_S3_NP2) PRIO=-1
;FOLD LIN Place_R1_L4_S3_NP2 CONT Vel=0.5 m/s LPlace_R1_L4_S3_NP2 Tool[2]:Lower Gripper Base[1]:Rack1;%{PE}%R8.3.21,%MKUKATPBASIS,%CMOVE,%VLIN,%P 1:LIN, 2:Place_R1_L4_S3_NP2, 3:C_DIS C_DIS, 5:0.5, 7:LPlace_R1_L4_S3_NP2
$BWDSTART=FALSE
LDAT_ACT= LLPlace_R1_L4_S3_NP2
FDAT_ACT= FPlace_R1_L4_S3_NP2
BAS(#CP_PARAMS,0.5)
LIN XPlace_R1_L4_S3_NP2 C_DIS C_DIS
;ENDFOLD
TRIGGER WHEN DISTANCE=1 DELAY=-1 DO Schrittmerker_R1Place(10300,10301,FPlace_R1_L4_S3_NP3,XPlace_R1_L4_S3_NP3) PRIO=-1
;FOLD LIN Place_R1_L4_S3_NP3 Vel=0.5 m/s LPlace_R1_L4_S3_NP3 Tool[2]:Lower Gripper Base[1]:Rack 1 ;%{PE}
$BWDSTART=FALSE
LDAT_ACT=LLPlace_R1_L4_S3_NP3
FDAT_ACT=FPlace_R1_L4_S3_NP3
BAS(#CP_PARAMS, 0.5)
LIN XPlace_R1_L4_S3_NP3
;ENDFOLD
TRIGGER WHEN DISTANCE=1 DELAY=-1 DO Schrittmerker_R1Place(10301,10302,FPlace_R1_L4_S3_NP4,XPlace_R1_L4_S3_NP4) PRIO=-1
;FOLD PTP Place_R1_L4_S3_NP4 CONT Vel=100 % PPlace_R1_L4_S3_NP4 Tool[2]:Lower Gripper Base[0];%{PE}%R8.3.21,%MKUKATPBASIS,%CMOVE,%VPTP,%P 1:PTP, 2:Place_R1_L4_S3_NP4, 3:C_DIS, 5:100, 7:PPlace_R1_L4_S3_NP4
$BWDSTART=FALSE
PDAT_ACT= PPPlace_R1_L4_S3_NP4
FDAT_ACT= FPlace_R1_L4_S3_NP4
BAS(#PTP_PARAMS,100)
PTP XPlace_R1_L4_S3_NP4 C_DIS
;ENDFOLD
TRIGGER WHEN DISTANCE=1 DELAY=-1 DO Schrittmerker_R1Place(10302,10303,FPlace_R1_L4_S3_NP5,XPlace_R1_L4_S3_NP5) PRIO=-1
;FOLD PTP Place_R1_L4_S3_NP5 CONT Vel=100 % PPlace_R1_L4_S3_NP5 Tool[2]:Lower Gripper Base[0];%{PE}%R8.3.21,%MKUKATPBASIS,%CMOVE,%VPTP,%P 1:PTP, 2:Place_R1_L4_S3_NP5, 3:C_DIS, 5:100, 7:PPlace_R1_L4_S3_NP5
$BWDSTART=FALSE
PDAT_ACT= PPPlace_R1_L4_S3_NP5
FDAT_ACT= FPlace_R1_L4_S3_NP5
BAS(#PTP_PARAMS,100)
PTP XPlace_R1_L4_S3_NP5 C_DIS
;ENDFOLD
TRIGGER WHEN DISTANCE=1 DELAY=-1 DO Schrittmerker_R1Place(10303,10304,FPlace_R1_L4_S3_NP6,XPlace_R1_L4_S3_NP6) PRIO=-1
;FOLD PTP Place_R1_L4_S3_NP6 CONT Vel=100 % PPlace_R1_L4_S3_NP6 Tool[2]:Lower Gripper Base[0];%{PE}%R8.3.21,%MKUKATPBASIS,%CMOVE,%VPTP,%P 1:PTP, 2:Place_R1_L4_S3_NP6, 3:C_DIS, 5:100, 7:PPlace_R1_L4_S3_NP6
$BWDSTART=FALSE
PDAT_ACT= PPPlace_R1_L4_S3_NP6
FDAT_ACT= FPlace_R1_L4_S3_NP6
BAS(#PTP_PARAMS,100)
PTP XPlace_R1_L4_S3_NP6 C_DIS
;ENDFOLD
TRIGGER WHEN DISTANCE=1 DELAY=-1 DO Schrittmerker_R1Place(10304,10305,FPlace_R1_L4_S3_NP7,XPlace_R1_L4_S3_NP7) PRIO=-1
;FOLD PTP Place_R1_L4_S3_NP7 CONT Vel=100 % PPlace_R1_L4_S3_NP7 Tool[2]:Lower Gripper Base[0];%{PE}
;FOLD Parameters ;%{h}
;Params IlfProvider=kukaroboter.basistech.inlineforms.movement.old; Kuka.IsGlobalPoint=False; Kuka.PointName=Place_R1_L4_S3_NP7; Kuka.BlendingEnabled=True; Kuka.MoveDataPtpName=PPlace_R1_L4_S3_NP7; Kuka.VelocityPtp=100; Kuka.CurrentCDSetIndex=0; Kuka.MovementParameterFieldEnabled=True; IlfCommand=PTP
;ENDFOLD
$BWDSTART = FALSE
PDAT_ACT = PPPlace_R1_L4_S3_NP7
FDAT_ACT = FPlace_R1_L4_S3_NP7
BAS(#PTP_PARAMS, 100.0)
SET_CD_PARAMS (0)
PTP XPlace_R1_L4_S3_NP7 C_Dis
;ENDFOLD

TRIGGER WHEN DISTANCE=1 DELAY=-1 DO Schrittmerker_R1Place(10305,10002,FHOME1,$nullframe,XHOME1) PRIO=-1
;FOLD PTP HOME1 Vel=100 % PHome1;%{PE}%R8.3.21,%MKUKATPBASIS,%CMOVE,%VPTP,%P 1:PTP, 2:HOME1, 3:, 5:100, 7:PHome1
$BWDSTART=FALSE
PDAT_ACT= PPHome1
FDAT_ACT= FHOME1
BAS(#PTP_PARAMS,100)
PTP XHOME1
;ENDFOLD

;***************************************************
;FOLD Final tasks.
; Robot out of area Rack 1 Level 4
RobAusStorage1_4_A70=RESET_IN_AREA
;***************************************************
; stop cyclic clearence check
$CYCFLAG[ciFreigabeSPS]=DISABLE_MONITORING
;***************************************************
; Disable collision detection
;FOLD COLLDETECT Off ;%{PE}
;FOLD Parameters ;%{h}
;Params IlfProvider=kukaroboter.basistech.inlineforms.colldetect.off; CollDetect.Command=Off
;ENDFOLD
USE_CD_PARAMS(0)
;ENDFOLD
;***************************************************
;ENDFOLD
;***************************************************

END

; ##################################################

GLOBAL DEF UP_Place_R1_L4_S4( )
;***************************************************
; Place part on:
;    Rack  1
;    Level 4
;    Shelf 4
;***************************************************
;FOLD Preconditions - Vorraussetzungen
;***************************************************
; Enable collision detection
;FOLD COLLDETECT SetLimits Axis1: 150 % Axis2: 200 % Axis3: 150 % Axis4: 200 % Axis5: 150 % Axis6: 150 % ;%{PE}
;FOLD Parameters ;%{h}
;Params IlfProvider=kukaroboter.basistech.inlineforms.colldetect.setlimits; CollDetect.Command=SetLimits; CollDetect.Axis1=150; CollDetect.Axis2=200; CollDetect.Axis3=150; CollDetect.Axis4=200; CollDetect.Axis5=150; CollDetect.Axis6=150
;ENDFOLD
SET_TQ_VALUES(150, 200, 150, 200, 150, 150)
;ENDFOLD
;***************************************************
; Check for part in gripper (tool 2).
CheckPartPresent(OCCUPIED_GRIPPER,PART_ON_TOOL_2)
;***************************************************
; Enable part lost detection for tool 2
SetPartLostDetection(PART_ON_TOOL_2)
;***************************************************
; Set load data.
SetLoadData( )
;***************************************************
; Robot has to start from home position.
IF NOT $IN_HOME1 THEN
  UP_HomeToHome(1)
ENDIF
;***************************************************
;ENDFOLD

TRIGGER WHEN DISTANCE=1 DELAY=-1 DO Schrittmerker_R1Place(10002,10002,FHOME1,$nullframe,XHOME1) PRIO=-1
;FOLD PTP HOME1 Vel=12 % PHome1;%{PE}%R8.3.21,%MKUKATPBASIS,%CMOVE,%VPTP,%P 1:PTP, 2:HOME1, 3:, 5:12, 7:PHome1
$BWDSTART=FALSE
PDAT_ACT= PPHome1
FDAT_ACT= FHOME1
BAS(#PTP_PARAMS,12)
PTP XHOME1
;ENDFOLD

;***************************************************
;FOLD Area clearence handshake.
IF NOT $FLAG[M_Inbetriebnahme] THEN
  ;-------------------------------------------------
  ; Request area clearence.
  AnfStoer_Store1_4_A102=SET_REQUEST
  ;-------------------------------------------------
  ; Wait for area clearence from PLC.
  WAIT_FOR_INPUT("Frg_Storage1_4_E70",TRUE)
  ;-------------------------------------------------
  ; Reset area clearence request.
  AnfStoer_Store1_4_A102=RESET_REQUEST
  ;-------------------------------------------------
  ; start cyclic clearence check
  $CYCFLAG[ciFreigabeSPS]=Frg_Storage1_4_E70
  ;-------------------------------------------------
ENDIF
;***************************************************
; set "robot in area"
RobAusStorage1_4_A70=SET_IN_AREA
;ENDFOLD
;***************************************************

;***************************************************
;FOLD Check for Teachmode
IF $FLAG[M_Teachen] THEN
  WAIT FOR $T1
ENDIF
;ENDFOLD
;***************************************************

